KUKA KRL program: MyProgram_155().src

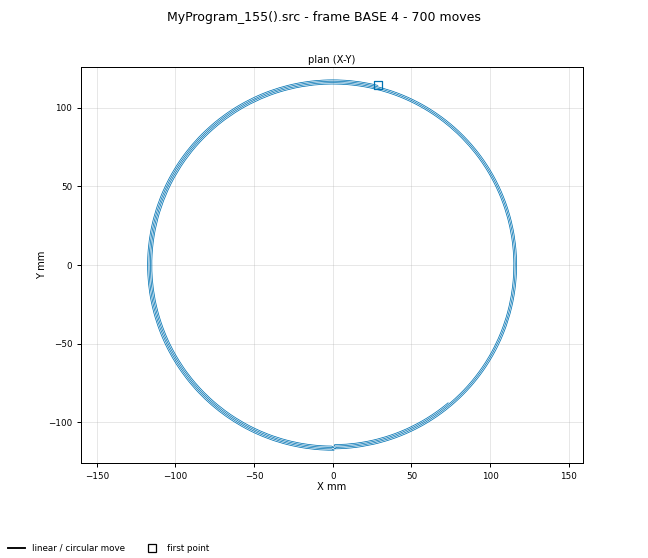
[picture p0: tool path of MyProgram_155().src in frame BASE 4, 700 of 700 moves have a stored position in this frame; points joined in program order, loops and branches not executed]
&ACCESS RVP
&REL 1
&PARAM TEMPLATE = C:\KRC\Roboter\Template\vorgabe
&PARAM EDITMASK = *
DEF MyProgram_155()
; ---- Setting reference (Base) ----
$BASE = BASE_DATA[4]

; --------------------------
; ---- Setting tool (TCP) ----
$TOOL = TOOL_DATA[3]
; --------------------------

$VEL.CP = VEL_APROX_PRINT
Startdeposition()
$VEL.CP = VEL_PRINT
LIN {X 28.6075,Y 114.2074,Z 120,A 72.0613,B 24.9358,C -1.85,E1 25.0377,E2 373.8713} C_DIS
LIN {X 25.7961,Y 114.8751,Z 120,A 73.4659,B 24.9358,C -1.8507,E1 25.0339,E2 372.4669} C_DIS
LIN {X 22.9691,Y 115.4736,Z 120,A 74.8709,B 24.9358,C -1.8512,E1 25.03,E2 371.0624} C_DIS
LIN {X 19.9429,Y 116.0335,Z 120,A 76.3004,B 24.9359,C -1.8487,E1 25.0261,E2 369.6403} C_DIS
LIN {X 17.2754,Y 116.4615,Z 120,A 77.5817,B 24.936,C -1.8476,E1 25.0226,E2 368.3629} C_DIS
LIN {X 14.0119,Y 116.8973,Z 120,A 79.1444,B 24.9361,C -1.8462,E1 25.0183,E2 366.8047} C_DIS
LIN {X 11.5401,Y 117.1689,Z 120,A 80.3543,B 24.9361,C -1.8463,E1 25.0149,E2 365.5954} C_DIS
LIN {X 8.2592,Y 117.444,Z 120,A 81.7792,B 24.9366,C -1.8385,E1 25.011,E2 364.1898} C_DIS
LIN {X 5.3745,Y 117.6113,Z 120,A 83.363,B 24.9361,C -1.8464,E1 25.0065,E2 362.5878} C_DIS
LIN {X 2.8894,Y 117.7004,Z 120,A 84.5732,B 24.9361,C -1.8462,E1 25.0032,E2 361.3782} C_DIS
LIN {X -0.4029,Y 117.7334,Z 120,A 85.999,B 24.9367,C -1.8381,E1 24.9992,E2 359.9717} C_DIS
LIN {X -3.2921,Y 117.688,Z 120,A 87.6216,B 24.936,C -1.8474,E1 24.9946,E2 358.3271} C_DIS
LIN {X -6.1794,Y 117.5718,Z 120,A 88.9298,B 24.9364,C -1.8425,E1 24.991,E2 357.03} C_DIS
LIN {X -9.0628,Y 117.3847,Z 120,A 90.3978,B 24.9362,C -1.8447,E1 24.9869,E2 355.5564} C_DIS
LIN {X -11.5401,Y 117.1689,Z 120,A 91.6095,B 24.9362,C -1.8441,E1 24.9835,E2 354.3454} C_DIS
LIN {X -14.4121,Y 116.8504,Z 120,A 93.1564,B 24.9359,C -1.8495,E1 24.9792,E2 352.7847} C_DIS
LIN {X -17.2754,Y 116.4615,Z 120,A 94.5644,B 24.9359,C -1.8486,E1 24.9753,E2 351.3776} C_DIS
LIN {X -20.1283,Y 116.0025,Z 120,A 95.973,B 24.936,C -1.8477,E1 24.9715,E2 349.9698} C_DIS
LIN {X -22.9691,Y 115.4736,Z 120,A 97.3817,B 24.936,C -1.8467,E1 24.9676,E2 348.5621} C_DIS
LIN {X -25.7961,Y 114.8751,Z 120,A 98.7906,B 24.9362,C -1.8455,E1 24.9638,E2 347.1541} C_DIS
LIN {X -28.6075,Y 114.2074,Z 120,A 100.1998,B 24.9362,C -1.8443,E1 24.9599,E2 345.7459} C_DIS
LIN {X -31.7893,Y 113.3611,Z 120,A 101.667,B 24.9368,C -1.8367,E1 24.956,E2 344.2943} C_DIS
LIN {X -34.1769,Y 112.6662,Z 120,A 103.0191,B 24.9364,C -1.8415,E1 24.9524,E2 342.9286} C_DIS
LIN {X -37.0459,Y 111.7549,Z 120,A 104.2953,B 24.9371,C -1.8316,E1 24.949,E2 341.6737} C_DIS
LIN {X -39.664,Y 110.8535,Z 120,A 105.7247,B 24.937,C -1.8334,E1 24.9453,E2 340.2371} C_DIS
LIN {X -42.3725,Y 109.8467,Z 120,A 107.2493,B 24.9368,C -1.8367,E1 24.9413,E2 338.7016} C_DIS
LIN {X -45.0555,Y 108.7737,Z 120,A 108.5208,B 24.9373,C -1.8288,E1 24.938,E2 337.4459} C_DIS
LIN {X -47.7114,Y 107.6352,Z 120,A 109.9314,B 24.9374,C -1.8269,E1 24.9344,E2 336.0364} C_DIS
LIN {X -50.68,Y 106.2678,Z 120,A 111.5717,B 24.9374,C -1.8266,E1 24.9302,E2 334.3928} C_DIS
LIN {X -53.2942,Y 104.9811,Z 120,A 112.9504,B 24.9377,C -1.8226,E1 24.9268,E2 333.0199} C_DIS
LIN {X -55.5003,Y 103.8337,Z 120,A 114.1649,B 24.9379,C -1.8207,E1 24.9238,E2 331.8065} C_DIS
LIN {X -58.0318,Y 102.4404,Z 120,A 115.5766,B 24.938,C -1.8185,E1 24.9204,E2 330.396} C_DIS
LIN {X -60.5283,Y 100.9854,Z 120,A 116.9884,B 24.9382,C -1.8162,E1 24.917,E2 328.9855} C_DIS
LIN {X -62.9884,Y 99.4695,Z 120,A 118.4003,B 24.9383,C -1.8138,E1 24.9137,E2 327.5749} C_DIS
LIN {X -65.4105,Y 97.8938,Z 120,A 119.9516,B 24.9381,C -1.8172,E1 24.91,E2 326.0103} C_DIS
LIN {X -68.1213,Y 96.025,Z 120,A 121.4219,B 24.9387,C -1.8083,E1 24.9067,E2 324.5561} C_DIS
LIN {X -70.4573,Y 94.3243,Z 120,A 122.8343,B 24.9389,C -1.8057,E1 24.9035,E2 323.145} C_DIS
LIN {X -72.4348,Y 92.8166,Z 120,A 124.0501,B 24.939,C -1.8033,E1 24.9008,E2 321.9305} C_DIS
LIN {X -74.6908,Y 91.011,Z 120,A 125.4632,B 24.9392,C -1.8005,E1 24.8978,E2 320.5187} C_DIS
LIN {X -76.9018,Y 89.1506,Z 120,A 126.8762,B 24.9394,C -1.7976,E1 24.8948,E2 319.1072} C_DIS
LIN {X -79.3634,Y 86.9641,Z 120,A 128.3082,B 24.9402,C -1.7867,E1 24.8918,E2 317.6952} C_DIS
LIN {X -81.1836,Y 85.2698,Z 120,A 129.7028,B 24.9398,C -1.7916,E1 24.889,E2 316.2833} C_DIS
LIN {X -83.2518,Y 83.2518,Z 120,A 131.2559,B 24.9397,C -1.7944,E1 24.8859,E2 314.7171} C_DIS
LIN {X -85.2976,Y 81.1541,Z 120,A 132.6747,B 24.9399,C -1.7905,E1 24.8831,E2 313.3013} C_DIS
LIN {X -87.5053,Y 78.7663,Z 120,A 134.1381,B 24.9405,C -1.7815,E1 24.8804,E2 311.8529} C_DIS
LIN {X -89.1506,Y 76.9018,Z 120,A 135.4975,B 24.9403,C -1.7846,E1 24.8779,E2 310.4799} C_DIS
LIN {X -91.2647,Y 74.3778,Z 120,A 136.9698,B 24.941,C -1.7749,E1 24.8753,E2 309.0239} C_DIS
LIN {X -92.8166,Y 72.4348,Z 120,A 138.1869,B 24.9412,C -1.772,E1 24.8732,E2 307.8081} C_DIS
LIN {X -94.5663,Y 70.1351,Z 120,A 139.7409,B 24.941,C -1.7743,E1 24.8706,E2 306.2411} C_DIS
LIN {X -96.259,Y 67.7932,Z 120,A 141.0161,B 24.9416,C -1.7649,E1 24.8685,E2 304.982} C_DIS
LIN {X -97.8938,Y 65.4105,Z 120,A 142.5702,B 24.9415,C -1.7672,E1 24.8661,E2 303.4147} C_DIS
LIN {X -99.4695,Y 62.9884,Z 120,A 143.9852,B 24.9417,C -1.7635,E1 24.864,E2 302.0013} C_DIS
LIN {X -101.1904,Y 60.1814,Z 120,A 145.2797,B 24.9429,C -1.7461,E1 24.8621,E2 300.7417} C_DIS
LIN {X -102.4404,Y 58.0318,Z 120,A 146.8155,B 24.9422,C -1.7561,E1 24.86,E2 299.1741} C_DIS
LIN {X -104.1352,Y 54.9278,Z 120,A 148.336,B 24.9431,C -1.7427,E1 24.858,E2 297.6775} C_DIS
LIN {X -105.8265,Y 51.5985,Z 120,A 150.2163,B 24.9433,C -1.7398,E1 24.8556,E2 295.7939} C_DIS
LIN {X -107.0416,Y 49.0287,Z 120,A 151.6575,B 24.9433,C -1.738,E1 24.8539,E2 294.3491} C_DIS
LIN {X -108.2126,Y 46.387,Z 120,A 153.1846,B 24.9433,C -1.7387,E1 24.8522,E2 292.8119} C_DIS
LIN {X -109.4657,Y 43.3423,Z 120,A 154.4796,B 24.9445,C -1.721,E1 24.8509,E2 291.5518} C_DIS
LIN {X -110.5368,Y 40.5322,Z 120,A 155.9008,B 24.9449,C -1.7147,E1 24.8495,E2 290.1376} C_DIS
LIN {X -111.3319,Y 38.3007,Z 120,A 157.3984,B 24.9442,C -1.7254,E1 24.8481,E2 288.6062} C_DIS
LIN {X -112.2383,Y 35.5569,Z 120,A 158.7082,B 24.9448,C -1.7169,E1 24.847,E2 287.309} C_DIS
LIN {X -113.2232,Y 32.2759,Z 120,A 160.3455,B 24.9452,C -1.7104,E1 24.8457,E2 285.6778} C_DIS
LIN {X -113.9481,Y 29.6166,Z 120,A 161.559,B 24.9458,C -1.7008,E1 24.8448,E2 284.48} C_DIS
LIN {X -114.5499,Y 27.2038,Z 120,A 163.0954,B 24.9452,C -1.7104,E1 24.8438,E2 282.9118} C_DIS
LIN {X -115.264,Y 23.9897,Z 120,A 164.3908,B 24.9463,C -1.6926,E1 24.8431,E2 281.6513} C_DIS
LIN {X -115.8181,Y 21.1538,Z 120,A 165.807,B 24.9466,C -1.6884,E1 24.8423,E2 280.2367} C_DIS
LIN {X -116.3023,Y 18.3051,Z 120,A 167.2233,B 24.9468,C -1.6843,E1 24.8417,E2 278.8218} C_DIS
LIN {X -116.6647,Y 15.845,Z 120,A 168.7598,B 24.9462,C -1.6938,E1 24.8411,E2 277.2534} C_DIS
LIN {X -117.0604,Y 12.5763,Z 120,A 170.0553,B 24.9474,C -1.6759,E1 24.8407,E2 275.9928} C_DIS
LIN {X -117.3017,Y 10.1014,Z 120,A 171.5922,B 24.9468,C -1.6855,E1 24.8403,E2 274.4239} C_DIS
LIN {X -117.5143,Y 7.2196,Z 120,A 173.0082,B 24.947,C -1.6813,E1 24.84,E2 273.0094} C_DIS
LIN {X -117.656,Y 4.3335,Z 120,A 174.4245,B 24.9473,C -1.6771,E1 24.8399,E2 271.5945} C_DIS
LIN {X -117.7313,Y 0.8208,Z 120,A 176.0503,B 24.9479,C -1.6681,E1 24.8398,E2 269.9803} C_DIS
LIN {X -117.7004,Y -2.8894,Z 120,A 177.825,B 24.9483,C -1.6609,E1 24.8398,E2 268.2121} C_DIS
LIN {X -117.5718,Y -6.1794,Z 120,A 179.2603,B 24.9491,C -1.6488,E1 24.84,E2 266.797} C_DIS
LIN {X -117.3847,Y -9.0628,Z 120,A -179.1455,B 24.9489,C -1.6521,E1 24.8403,E2 265.1855} C_DIS
LIN {X -117.1689,Y -11.5401,Z 120,A -177.9267,B 24.9491,C -1.6485,E1 24.8407,E2 263.9679} C_DIS
LIN {X -116.7986,Y -14.8117,Z 120,A -176.3132,B 24.9494,C -1.6439,E1 24.8412,E2 262.3558} C_DIS
LIN {X -116.4615,Y -17.2754,Z 120,A -174.9554,B 24.9492,C -1.6461,E1 24.8418,E2 260.9845} C_DIS
LIN {X -116.0025,Y -20.1283,Z 120,A -173.5394,B 24.9495,C -1.6421,E1 24.8424,E2 259.5697} C_DIS
LIN {X -115.4736,Y -22.9691,Z 120,A -172.1236,B 24.9497,C -1.638,E1 24.8432,E2 258.1553} C_DIS
LIN {X -114.7514,Y -26.3313,Z 120,A -170.5534,B 24.9503,C -1.6285,E1 24.8441,E2 256.5985} C_DIS
LIN {X -113.7427,Y -30.3958,Z 120,A -168.5264,B 24.9507,C -1.6217,E1 24.8455,E2 254.5758} C_DIS
LIN {X -112.9625,Y -33.178,Z 120,A -167.2894,B 24.9514,C -1.6104,E1 24.8464,E2 253.3588} C_DIS
LIN {X -112.1142,Y -35.9403,Z 120,A -165.8738,B 24.9516,C -1.6065,E1 24.8476,E2 251.9444} C_DIS
LIN {X -111.3319,Y -38.3007,Z 120,A -164.4772,B 24.9514,C -1.6106,E1 24.8489,E2 250.53} C_DIS
LIN {X -110.3584,Y -41.0214,Z 120,A -163.062,B 24.9516,C -1.6067,E1 24.8502,E2 249.1159} C_DIS
LIN {X -109.3184,Y -43.7173,Z 120,A -161.5073,B 24.9516,C -1.6088,E1 24.8518,E2 247.5475} C_DIS
LIN {X -108.2126,Y -46.387,Z 120,A -160.2317,B 24.9521,C -1.5993,E1 24.8532,E2 246.2877} C_DIS
LIN {X -107.0416,Y -49.0287,Z 120,A -158.8168,B 24.9523,C -1.5956,E1 24.8548,E2 244.8738} C_DIS
LIN {X -105.8062,Y -51.6408,Z 120,A -157.2625,B 24.9522,C -1.5978,E1 24.8567,E2 243.3057} C_DIS
LIN {X -104.3192,Y -54.5784,Z 120,A -155.9681,B 24.9532,C -1.5804,E1 24.8584,E2 242.0459} C_DIS
LIN {X -102.9484,Y -57.1221,Z 120,A -154.5537,B 24.9534,C -1.5769,E1 24.8602,E2 240.6325} C_DIS
LIN {X -101.7206,Y -59.2845,Z 120,A -152.9791,B 24.9527,C -1.5889,E1 24.8625,E2 239.0209} C_DIS
LIN {X -99.4695,Y -62.9884,Z 120,A -150.8974,B 24.9531,C -1.5822,E1 24.8655,E2 236.9446} C_DIS
LIN {X -97.6678,Y -65.7442,Z 120,A -149.4255,B 24.9537,C -1.5725,E1 24.8678,E2 235.4884} C_DIS
LIN {X -96.025,Y -68.1213,Z 120,A -148.0114,B 24.9539,C -1.5693,E1 24.8701,E2 234.075} C_DIS
LIN {X -94.3243,Y -70.4573,Z 120,A -146.5978,B 24.954,C -1.5661,E1 24.8724,E2 232.6622} C_DIS
LIN {X -92.8166,Y -72.4348,Z 120,A -145.3812,B 24.9542,C -1.5634,E1 24.8745,E2 231.4463} C_DIS
LIN {X -91.011,Y -74.6908,Z 120,A -143.8283,B 24.954,C -1.5663,E1 24.8772,E2 229.8793} C_DIS
LIN {X -88.8855,Y -77.2053,Z 120,A -142.5354,B 24.955,C -1.5494,E1 24.8795,E2 228.6207} C_DIS
LIN {X -87.2365,Y -79.0665,Z 120,A -141.0019,B 24.9544,C -1.5604,E1 24.8824,E2 227.0541} C_DIS
LIN {X -85.2698,Y -81.1836,Z 120,A -139.7283,B 24.9549,C -1.5516,E1 24.8849,E2 225.7959} C_DIS
LIN {X -82.9651,Y -83.535,Z 120,A -138.1185,B 24.9551,C -1.5485,E1 24.888,E2 224.1866} C_DIS
LIN {X -81.1836,Y -85.2698,Z 120,A -136.7639,B 24.9549,C -1.5522,E1 24.8908,E2 222.8176} C_DIS
LIN {X -78.7439,Y -87.5253,Z 120,A -135.4704,B 24.9559,C -1.535,E1 24.8934,E2 221.5598} C_DIS
LIN {X -76.8519,Y -89.1932,Z 120,A -133.931,B 24.9552,C -1.546,E1 24.8967,E2 219.9882} C_DIS
LIN {X -74.3778,Y -91.2647,Z 120,A -132.4694,B 24.9557,C -1.5384,E1 24.8998,E2 218.5392} C_DIS
LIN {X -72.2665,Y -92.9463,Z 120,A -131.2444,B 24.956,C -1.5321,E1 24.9025,E2 217.3247} C_DIS
LIN {X -70.1351,Y -94.5663,Z 120,A -129.7144,B 24.9556,C -1.5396,E1 24.9059,E2 215.7712} C_DIS
LIN {X -67.7933,Y -96.259,Z 120,A -128.4312,B 24.956,C -1.5319,E1 24.9088,E2 214.5021} C_DIS
LIN {X -65.3554,Y -97.9301,Z 120,A -126.873,B 24.9559,C -1.5348,E1 24.9125,E2 212.9318} C_DIS
LIN {X -62.9884,Y -99.4695,Z 120,A -125.6092,B 24.9563,C -1.5278,E1 24.9154,E2 211.6806} C_DIS
LIN {X -60.1814,Y -101.1904,Z 120,A -124.0018,B 24.9563,C -1.5257,E1 24.9193,E2 210.0732} C_DIS
LIN {X -57.994,Y -102.4615,Z 120,A -122.6437,B 24.9562,C -1.5295,E1 24.9226,E2 208.7021} C_DIS
LIN {X -55.5003,Y -103.8337,Z 120,A -121.3776,B 24.9566,C -1.5223,E1 24.9257,E2 207.4494} C_DIS
LIN {X -52.5743,Y -105.3435,Z 120,A -119.771,B 24.9566,C -1.5205,E1 24.9297,E2 205.8427} C_DIS
LIN {X -49.9732,Y -106.602,Z 120,A -118.361,B 24.9568,C -1.519,E1 24.9332,E2 204.4328} C_DIS
LIN {X -47.342,Y -107.7963,Z 120,A -117.1289,B 24.9573,C -1.5098,E1 24.9363,E2 203.2196} C_DIS
LIN {X -44.6823,Y -108.9256,Z 120,A -115.5421,B 24.9569,C -1.5163,E1 24.9404,E2 201.6138} C_DIS
LIN {X -41.8052,Y -110.0615,Z 120,A -114.0944,B 24.9572,C -1.5123,E1 24.9442,E2 200.1724} C_DIS
LIN {X -39.2838,Y -110.9869,Z 120,A -112.724,B 24.9571,C -1.5139,E1 24.9478,E2 198.7955} C_DIS
LIN {X -36.9316,Y -111.7935,Z 120,A -111.3729,B 24.9568,C -1.5192,E1 24.9514,E2 197.4294} C_DIS
LIN {X -33.9916,Y -112.7211,Z 120,A -109.9455,B 24.957,C -1.5148,E1 24.9552,E2 196.0098} C_DIS
LIN {X -31.4016,Y -113.471,Z 120,A -108.5562,B 24.9569,C -1.5174,E1 24.959,E2 194.6122} C_DIS
LIN {X -28.6075,Y -114.2074,Z 120,A -107.1484,B 24.9569,C -1.5166,E1 24.9628,E2 193.2041} C_DIS
LIN {X -25.7961,Y -114.8751,Z 120,A -105.7406,B 24.9569,C -1.516,E1 24.9666,E2 191.7961} C_DIS
LIN {X -22.9691,Y -115.4736,Z 120,A -104.3331,B 24.9569,C -1.5155,E1 24.9705,E2 190.3881} C_DIS
LIN {X -20.1283,Y -116.0025,Z 120,A -102.9258,B 24.9569,C -1.515,E1 24.9743,E2 188.9805} C_DIS
LIN {X -17.2754,Y -116.4615,Z 120,A -101.6573,B 24.9574,C -1.5084,E1 24.9778,E2 187.7265} C_DIS
LIN {X -14.0119,Y -116.8973,Z 120,A -100.0542,B 24.9574,C -1.5082,E1 24.9822,E2 186.1229} C_DIS
LIN {X -11.5401,Y -117.1689,Z 120,A -98.8438,B 24.9574,C -1.5081,E1 24.9856,E2 184.912} C_DIS
LIN {X -8.2592,Y -117.444,Z 120,A -97.3129,B 24.9576,C -1.5048,E1 24.9899,E2 183.3882} C_DIS
LIN {X -5.3745,Y -117.6113,Z 120,A -95.8351,B 24.9574,C -1.5082,E1 24.994,E2 181.9021} C_DIS
LIN {X -2.8894,Y -117.7004,Z 120,A -94.6255,B 24.9574,C -1.5082,E1 24.9974,E2 180.6921} C_DIS
LIN {X 0.8293,Y -117.7293,Z 120,A -93.0037,B 24.9578,C -1.5002,E1 25.0019,E2 179.0895} C_DIS
Enddeposition()
LIN {X 0.8293,Y -117.7293,Z 120,A -93.0037,B 24.9578,C -1.5002,E1 25.0019,E2 179.0895} C_DIS
Startdeposition()
$VEL.CP = VEL_PRINT
LIN {X -0.5833,Y -116.846,Z 120,A -94.2822,B 24.9585,C -1.4892,E1 24.9982,E2 180.394} C_DIS
LIN {X -3.7681,Y -116.7867,Z 120,A -95.7825,B 24.9583,C -1.4917,E1 24.994,E2 181.8886} C_DIS
LIN {X -6.6179,Y -116.6599,Z 120,A -97.1718,B 24.9583,C -1.492,E1 24.9902,E2 183.2775} C_DIS
LIN {X -9.8038,Y -116.4364,Z 120,A -98.8453,B 24.9586,C -1.4872,E1 24.9855,E2 184.963} C_DIS
LIN {X -13.6561,Y -116.0466,Z 120,A -100.6924,B 24.9584,C -1.4898,E1 24.9804,E2 186.8052} C_DIS
LIN {X -17.4959,Y -115.5306,Z 120,A -102.5961,B 24.9584,C -1.49,E1 24.9751,E2 188.7098} C_DIS
LIN {X -20.8591,Y -114.9706,Z 120,A -104.2133,B 24.9582,C -1.493,E1 24.9707,E2 190.3216} C_DIS
LIN {X -24.4922,Y -114.2524,Z 120,A -106.1589,B 24.9585,C -1.4881,E1 24.9653,E2 192.2812} C_DIS
LIN {X -27.6951,Y -113.5178,Z 120,A -107.672,B 24.9582,C -1.4932,E1 24.9612,E2 193.7841} C_DIS
LIN {X -30.8948,Y -112.6899,Z 120,A -109.1999,B 24.9579,C -1.4983,E1 24.9571,E2 195.3023} C_DIS
LIN {X -33.8766,Y -111.8301,Z 120,A -111.8951,B 24.9607,C -1.4487,E1 24.9496,E2 198.1197} C_DIS
LIN {X -40.072,Y -109.7613,Z 120,A -113.983,B 24.9579,C -1.4994,E1 24.9444,E2 200.0914} C_DIS
LIN {X -43.4727,Y -108.4612,Z 120,A -115.8418,B 24.9579,C -1.4979,E1 24.9395,E2 201.9578} C_DIS
LIN {X -47.2007,Y -106.8911,Z 120,A -117.7204,B 24.9576,C -1.5046,E1 24.9348,E2 203.8249} C_DIS
LIN {X -49.4784,Y -105.8548,Z 120,A -119.1132,B 24.9579,C -1.4989,E1 24.9312,E2 205.2347} C_DIS
LIN {X -53.1358,Y -104.0668,Z 120,A -120.8787,B 24.9572,C -1.5113,E1 24.9268,E2 206.9753} C_DIS
LIN {X -56.434,Y -102.3176,Z 120,A -122.7584,B 24.9572,C -1.5116,E1 24.9222,E2 208.8596} C_DIS
LIN {X -59.1122,Y -100.7929,Z 120,A -124.3925,B 24.9574,C -1.5085,E1 24.9182,E2 210.5059} C_DIS
LIN {X -61.827,Y -99.1501,Z 120,A -125.9835,B 24.9574,C -1.5094,E1 24.9144,E2 212.0998} C_DIS
LIN {X -65.022,Y -97.0865,Z 120,A -127.9181,B 24.9574,C -1.5094,E1 24.9099,E2 214.0408} C_DIS
LIN {X -68.4014,Y -94.7364,Z 120,A -130.2054,B 24.9578,C -1.5014,E1 24.9046,E2 216.3548} C_DIS
LIN {X -71.0173,Y -92.7901,Z 120,A -131.2356,B 24.9562,C -1.5284,E1 24.9025,E2 217.3248} C_DIS
LIN {X -73.512,Y -90.8256,Z 120,A -133.0468,B 24.9567,C -1.5205,E1 24.8985,E2 219.1614} C_DIS
LIN {X -76.9746,Y -87.9104,Z 120,A -135.1903,B 24.9563,C -1.528,E1 24.8939,E2 221.2953} C_DIS
LIN {X -79.5354,Y -85.6032,Z 120,A -136.9573,B 24.9563,C -1.5282,E1 24.8903,E2 223.0691} C_DIS
LIN {X -83.7073,Y -81.5277,Z 120,A -139.6988,B 24.9556,C -1.5392,E1 24.8849,E2 225.7958} C_DIS
LIN {X -86.2695,Y -78.8096,Z 120,A -141.6709,B 24.9557,C -1.5374,E1 24.8811,E2 227.7808} C_DIS
LIN {X -89.6384,Y -74.956,Z 120,A -144.2184,B 24.9555,C -1.5417,E1 24.8764,E2 230.3298} C_DIS
LIN {X -91.9256,Y -72.1328,Z 120,A -146.5553,B 24.9565,C -1.523,E1 24.8723,E2 232.7221} C_DIS
LIN {X -94.566,Y -68.6354,Z 120,A -148.019,B 24.9546,C -1.5567,E1 24.87,E2 234.1128} C_DIS
LIN {X -95.9693,Y -66.6574,Z 120,A -149.3147,B 24.9546,C -1.5553,E1 24.8679,E2 235.4182} C_DIS
LIN {X -98.1483,Y -63.406,Z 120,A -151.5108,B 24.9551,C -1.5488,E1 24.8645,E2 237.6406} C_DIS
LIN {X -100.0436,Y -60.3715,Z 120,A -153.0221,B 24.9542,C -1.5635,E1 24.8623,E2 239.1247} C_DIS
LIN {X -102.1243,Y -56.7802,Z 120,A -155.075,B 24.9539,C -1.5683,E1 24.8595,E2 241.1769} C_DIS
LIN {X -104.1156,Y -53.0403,Z 120,A -157.1484,B 24.9536,C -1.5743,E1 24.8568,E2 243.2472} C_DIS
LIN {X -105.5963,Y -50.0314,Z 120,A -158.9261,B 24.9536,C -1.5734,E1 24.8546,E2 245.0364} C_DIS
LIN {X -108.1129,Y -44.3283,Z 120,A -161.6818,B 24.9524,C -1.5946,E1 24.8516,E2 247.7568} C_DIS
LIN {X -108.9291,Y -42.2844,Z 120,A -162.8718,B 24.9524,C -1.5933,E1 24.8504,E2 248.9568} C_DIS
LIN {X -109.8159,Y -39.9223,Z 120,A -164.2194,B 24.9524,C -1.5924,E1 24.8491,E2 250.314} C_DIS
LIN {X -111.2193,Y -35.8272,Z 120,A -166.3646,B 24.9522,C -1.5979,E1 24.8472,E2 252.4583} C_DIS
LIN {X -112.4296,Y -31.8258,Z 120,A -168.4471,B 24.9519,C -1.6029,E1 24.8455,E2 254.541} C_DIS
LIN {X -113.5161,Y -27.702,Z 120,A -170.5072,B 24.9514,C -1.6106,E1 24.8441,E2 256.5947} C_DIS
LIN {X -114.2632,Y -24.4427,Z 120,A -172.1219,B 24.951,C -1.6167,E1 24.8431,E2 258.2043} C_DIS
LIN {X -114.9448,Y -21.0025,Z 120,A -173.8973,B 24.9508,C -1.6199,E1 24.8422,E2 259.9827} C_DIS
LIN {X -115.8291,Y -15.3974,Z 120,A -176.4915,B 24.9498,C -1.6364,E1 24.8411,E2 262.553} C_DIS
LIN {X -116.295,Y -11.3652,Z 120,A -178.8276,B 24.9503,C -1.6287,E1 24.8404,E2 264.9214} C_DIS
LIN {X -116.6596,Y -6.6243,Z 120,A 178.8642,B 24.9498,C -1.6372,E1 24.84,E2 267.2232} C_DIS
LIN {X -116.8144,Y -2.8659,Z 120,A 177.0384,B 24.9494,C -1.6439,E1 24.8398,E2 269.044} C_DIS
LIN {X -116.8438,Y 0.9933,Z 120,A 175.1495,B 24.949,C -1.6503,E1 24.8398,E2 270.9291} C_DIS
LIN {X -116.7276,Y 5.2971,Z 120,A 172.8004,B 24.9491,C -1.6476,E1 24.84,E2 273.2989} C_DIS
LIN {X -116.489,Y 9.1463,Z 120,A 171.1669,B 24.9481,C -1.6641,E1 24.8404,E2 274.9027} C_DIS
LIN {X -115.8711,Y 15.0729,Z 120,A 168.3215,B 24.9473,C -1.6767,E1 24.8413,E2 277.7351} C_DIS
LIN {X -115.1266,Y 19.9815,Z 120,A 165.8287,B 24.947,C -1.6822,E1 24.8423,E2 280.2296} C_DIS
LIN {X -114.6957,Y 22.3215,Z 120,A 164.015,B 24.9484,C -1.6599,E1 24.8433,E2 282.1071} C_DIS
LIN {X -113.8096,Y 26.4711,Z 120,A 161.8481,B 24.9482,C -1.6632,E1 24.8447,E2 284.2791} C_DIS
LIN {X -112.6767,Y 30.9437,Z 120,A 160.3303,B 24.9458,C -1.7004,E1 24.8457,E2 285.717} C_DIS
LIN {X -111.952,Y 33.4681,Z 120,A 158.9357,B 24.9458,C -1.7001,E1 24.8468,E2 287.1203} C_DIS
LIN {X -110.6888,Y 37.4339,Z 120,A 156.8632,B 24.9455,C -1.7053,E1 24.8486,E2 289.1923} C_DIS
LIN {X -109.648,Y 40.3826,Z 120,A 155.3478,B 24.9451,C -1.7108,E1 24.8501,E2 290.7031} C_DIS
LIN {X -108.6603,Y 42.9688,Z 120,A 153.8954,B 24.9451,C -1.7112,E1 24.8515,E2 292.1628} C_DIS
LIN {X -106.5918,Y 47.8697,Z 120,A 151.318,B 24.9445,C -1.7204,E1 24.8544,E2 294.7323} C_DIS
LIN {X -104.0815,Y 53.1071,Z 120,A 148.8034,B 24.9431,C -1.7426,E1 24.8574,E2 297.2078} C_DIS
LIN {X -102.348,Y 56.3794,Z 120,A 146.3255,B 24.9445,C -1.721,E1 24.8608,E2 299.7503} C_DIS
LIN {X -99.8932,Y 60.619,Z 120,A 144.2276,B 24.9432,C -1.7403,E1 24.8637,E2 301.8129} C_DIS
LIN {X -98.0409,Y 63.5734,Z 120,A 142.3789,B 24.9432,C -1.7395,E1 24.8665,E2 303.6729} C_DIS
LIN {X -95.9693,Y 66.6573,Z 120,A 140.6979,B 24.9426,C -1.7504,E1 24.8691,E2 305.3364} C_DIS
LIN {X -94.0429,Y 69.3499,Z 120,A 138.873,B 24.9428,C -1.7466,E1 24.8721,E2 307.1791} C_DIS
LIN {X -91.7233,Y 72.3888,Z 120,A 137.1219,B 24.9422,C -1.7567,E1 24.8751,E2 308.9144} C_DIS
LIN {X -89.8293,Y 74.7262,Z 120,A 135.7036,B 24.9417,C -1.763,E1 24.8776,E2 310.3244} C_DIS
LIN {X -87.5284,Y 77.4112,Z 120,A 133.9937,B 24.9414,C -1.7684,E1 24.8807,E2 312.0291} C_DIS
LIN {X -85.3016,Y 79.8562,Z 120,A 132.1845,B 24.9416,C -1.7648,E1 24.8842,E2 313.8548} C_DIS
LIN {X -82.6638,Y 82.586,Z 120,A 130.4757,B 24.9409,C -1.7756,E1 24.8875,E2 315.5452} C_DIS
LIN {X -80.9252,Y 84.288,Z 120,A 129.2342,B 24.9409,C -1.7765,E1 24.89,E2 316.7897} C_DIS
LIN {X -78.1093,Y 86.9039,Z 120,A 127.2894,B 24.9407,C -1.7785,E1 24.894,E2 318.7378} C_DIS
LIN {X -75.4686,Y 89.2074,Z 120,A 125.5023,B 24.9407,C -1.7795,E1 24.8978,E2 320.5293} C_DIS
LIN {X -72.6669,Y 91.5035,Z 120,A 123.7905,B 24.9402,C -1.7861,E1 24.9015,E2 322.2319} C_DIS
LIN {X -70.0802,Y 93.4991,Z 120,A 122.1557,B 24.9401,C -1.7881,E1 24.9051,E2 323.8678} C_DIS
LIN {X -67.4078,Y 95.4453,Z 120,A 120.6158,B 24.9396,C -1.7948,E1 24.9086,E2 325.3971} C_DIS
LIN {X -64.938,Y 97.1434,Z 120,A 119.1614,B 24.9394,C -1.7984,E1 24.912,E2 326.848} C_DIS
LIN {X -62.4604,Y 98.7544,Z 120,A 117.7195,B 24.9392,C -1.8015,E1 24.9153,E2 328.2871} C_DIS
LIN {X -59.4234,Y 100.609,Z 120,A 115.8698,B 24.9392,C -1.8003,E1 24.9198,E2 330.1451} C_DIS
LIN {X -56.786,Y 102.121,Z 120,A 114.3615,B 24.9392,C -1.8022,E1 24.9234,E2 331.6534} C_DIS
LIN {X -52.8753,Y 104.1999,Z 120,A 112.1336,B 24.939,C -1.8035,E1 24.929,E2 333.8843} C_DIS
LIN {X -45.1093,Y 107.7893,Z 120,A 107.9624,B 24.9385,C -1.8109,E1 24.9396,E2 338.0482} C_DIS
LIN {X -41.3286,Y 109.2943,Z 120,A 105.9734,B 24.9383,C -1.8139,E1 24.9447,E2 340.0344} C_DIS
LIN {X -38.0207,Y 110.4907,Z 120,A 104.1491,B 24.9385,C -1.8118,E1 24.9496,E2 341.8672} C_DIS
LIN {X -34.1404,Y 111.7496,Z 120,A 102.3429,B 24.9377,C -1.8224,E1 24.9543,E2 343.6513} C_DIS
LIN {X -31.8168,Y 112.4322,Z 120,A 101.0929,B 24.9378,C -1.821,E1 24.9577,E2 344.9066} C_DIS
LIN {X -28.5613,Y 113.3042,Z 120,A 99.1236,B 24.9386,C -1.8092,E1 24.9631,E2 346.9069} C_DIS
LIN {X -24.5198,Y 114.2464,Z 120,A 97.4082,B 24.9376,C -1.8247,E1 24.9677,E2 348.5877} C_DIS
LIN {X -20.8546,Y 114.9714,Z 120,A 95.5404,B 24.9376,C -1.8247,E1 24.9728,E2 350.4578} C_DIS
LIN {X -17.7549,Y 115.4906,Z 120,A 93.9865,B 24.9376,C -1.8252,E1 24.9771,E2 352.0118} C_DIS
LIN {X -13.8207,Y 116.0273,Z 120,A 91.9759,B 24.9376,C -1.8236,E1 24.9827,E2 354.0274} C_DIS
LIN {X -9.9632,Y 116.4237,Z 120,A 89.9577,B 24.9379,C -1.8195,E1 24.9883,E2 356.0565} C_DIS
LIN {X -6.0564,Y 116.691,Z 120,A 88.1401,B 24.9376,C -1.8247,E1 24.9933,E2 357.8624} C_DIS
LIN {X -1.865,Y 116.8328,Z 120,A 86.2333,B 24.9371,C -1.8318,E1 24.9986,E2 359.7526} C_DIS
LIN {X 0.9122,Y 116.844,Z 120,A 84.7627,B 24.9374,C -1.8273,E1 25.0028,E2 361.2337} C_DIS
LIN {X 4.2907,Y 116.7707,Z 120,A 83.2064,B 24.9371,C -1.8318,E1 25.0071,E2 362.779} C_DIS
LIN {X 7.6392,Y 116.5976,Z 120,A 81.5607,B 24.9371,C -1.8318,E1 25.0117,E2 364.4241} C_DIS
LIN {X 11.0317,Y 116.3258,Z 120,A 79.9381,B 24.937,C -1.8337,E1 25.0162,E2 366.0413} C_DIS
LIN {X 13.9759,Y 116.0092,Z 120,A 78.4496,B 24.9371,C -1.8318,E1 25.0203,E2 367.5332} C_DIS
LIN {X 17.163,Y 115.5821,Z 120,A 76.8742,B 24.9371,C -1.8314,E1 25.0246,E2 369.1081} C_DIS
LIN {X 20.0634,Y 115.1137,Z 120,A 75.4406,B 24.9371,C -1.8313,E1 25.0286,E2 370.5407} C_DIS
LIN {X 23.5374,Y 114.4522,Z 120,A 73.644,B 24.9374,C -1.8278,E1 25.0335,E2 372.3434} C_DIS
LIN {X 27.1678,Y 113.6464,Z 120,A 71.6794,B 24.9379,C -1.8205,E1 25.0389,E2 374.3224} C_DIS
LIN {X 31.2326,Y 112.5971,Z 120,A 68.7019,B 24.9407,C -1.7787,E1 25.0472,E2 377.3941} C_DIS
LIN {X 37.3634,Y 110.7126,Z 120,A 67.0087,B 24.9365,C -1.8405,E1 25.0513,E2 378.9378} C_DIS
LIN {X 41.4792,Y 109.2373,Z 120,A 64.5211,B 24.9377,C -1.823,E1 25.0579,E2 381.4616} C_DIS
LIN {X 44.7935,Y 107.9224,Z 120,A 62.8297,B 24.9377,C -1.8238,E1 25.0623,E2 383.1474} C_DIS
LIN {X 47.7574,Y 106.6424,Z 120,A 61.1868,B 24.938,C -1.8193,E1 25.0665,E2 384.7969} C_DIS
LIN {X 50.6964,Y 105.2767,Z 120,A 59.5747,B 24.9382,C -1.8164,E1 25.0706,E2 386.4118} C_DIS
LIN {X 54.3776,Y 103.4233,Z 120,A 57.5526,B 24.9383,C -1.8137,E1 25.0756,E2 388.4348} C_DIS
LIN {X 57.1544,Y 101.9153,Z 120,A 55.9552,B 24.9386,C -1.8093,E1 25.0795,E2 390.0378} C_DIS
LIN {X 59.9972,Y 100.2698,Z 120,A 54.47,B 24.9384,C -1.8126,E1 25.0831,E2 391.5107} C_DIS
LIN {X 62.2868,Y 98.8628,Z 120,A 52.9851,B 24.9391,C -1.803,E1 25.0866,E2 393.0136} C_DIS
LIN {X 65.5013,Y 96.762,Z 120,A 51.2606,B 24.9388,C -1.8071,E1 25.0906,E2 394.7225} C_DIS
LIN {X 68.9644,Y 94.3251,Z 120,A 49.171,B 24.9391,C -1.8029,E1 25.0954,E2 396.8147} C_DIS
LIN {X 71.7757,Y 92.2056,Z 120,A 47.3327,B 24.9396,C -1.7946,E1 25.0995,E2 398.6659} C_DIS
LIN {X 74.6746,Y 89.8722,Z 120,A 45.6175,B 24.9396,C -1.7962,E1 25.1031,E2 400.3709} C_DIS
LIN {X 77.4613,Y 87.484,Z 120,A 43.9093,B 24.9395,C -1.7968,E1 25.1067,E2 402.0709} C_DIS
LIN {X 79.9413,Y 85.2215,Z 120,A 42.0637,B 24.9403,C -1.7842,E1 25.1106,E2 403.9387} C_DIS
LIN {X 83.0621,Y 82.1827,Z 120,A 39.9987,B 24.9404,C -1.7829,E1 25.1146,E2 405.9981} C_DIS
LIN {X 86.1353,Y 78.9558,Z 120,A 37.9564,B 24.9404,C -1.7846,E1 25.1185,E2 408.0274} C_DIS
LIN {X 88.394,Y 76.4209,Z 120,A 36.1064,B 24.9411,C -1.7722,E1 25.122,E2 409.8986} C_DIS
LIN {X 90.883,Y 73.4412,Z 120,A 34.3936,B 24.9408,C -1.7765,E1 25.125,E2 411.5932} C_DIS
LIN {X 92.7846,Y 71.0244,Z 120,A 32.9119,B 24.941,C -1.7741,E1 25.1275,E2 413.0737} C_DIS
LIN {X 94.5189,Y 68.6997,Z 120,A 31.4706,B 24.9413,C -1.7696,E1 25.1299,E2 414.5186} C_DIS
LIN {X 96.2888,Y 66.1978,Z 120,A 29.9752,B 24.9415,C -1.7661,E1 25.1323,E2 416.015} C_DIS
LIN {X 98.2987,Y 63.1718,Z 120,A 28.1702,B 24.9419,C -1.7604,E1 25.1351,E2 417.8245} C_DIS
LIN {X 100.0635,Y 60.3388,Z 120,A 26.4162,B 24.9426,C -1.7505,E1 25.1377,E2 419.5929} C_DIS
LIN {X 102.1404,Y 56.7513,Z 120,A 24.5377,B 24.9425,C -1.7522,E1 25.1402,E2 421.4576} C_DIS
LIN {X 103.7357,Y 53.7836,Z 120,A 22.7222,B 24.9433,C -1.7399,E1 25.1426,E2 423.2926} C_DIS
LIN {X 105.5627,Y 50.1012,Z 120,A 20.8355,B 24.9433,C -1.7402,E1 25.1449,E2 425.1684} C_DIS
LIN {X 107.0832,Y 46.76,Z 120,A 19.0772,B 24.9435,C -1.737,E1 25.1469,E2 426.9246} C_DIS
LIN {X 108.3952,Y 43.6347,Z 120,A 17.3018,B 24.9441,C -1.7268,E1 25.1488,E2 428.7145} C_DIS
LIN {X 109.831,Y 39.8808,Z 120,A 15.4704,B 24.9441,C -1.7275,E1 25.1506,E2 430.5339} C_DIS
LIN {X 111.0216,Y 36.4382,Z 120,A 13.6818,B 24.9444,C -1.7219,E1 25.1522,E2 432.3255} C_DIS
LIN {X 112.6061,Y 31.2032,Z 120,A 11.0755,B 24.9447,C -1.7173,E1 25.1543,E2 434.9279} C_DIS
LIN {X 113.4315,Y 28.0487,Z 120,A 9.3537,B 24.9454,C -1.7065,E1 25.1554,E2 436.6651} C_DIS
LIN {X 114.629,Y 22.668,Z 120,A 6.8322,B 24.9454,C -1.7065,E1 25.1569,E2 439.1718} C_DIS
LIN {X 115.2494,Y 19.2584,Z 120,A 5.1751,B 24.9456,C -1.7032,E1 25.1577,E2 440.8271} C_DIS
LIN {X 115.736,Y 16.0814,Z 120,A 3.5366,B 24.9461,C -1.6952,E1 25.1584,E2 442.4749} C_DIS
LIN {X 116.0749,Y 13.4148,Z 120,A 2.1386,B 24.9467,C -1.6872,E1 25.1589,E2 443.8835} C_DIS
LIN {X 116.4326,Y 9.8516,Z 120,A 0.333,B 24.9472,C -1.6791,E1 25.1593,E2 445.6974} C_DIS
LIN {X 116.706,Y 5.7829,Z 120,A -1.5154,B 24.9472,C -1.6798,E1 25.1596,E2 447.5332} C_DIS
LIN {X 116.8262,Y 2.2252,Z 120,A -3.2494,B 24.9474,C -1.6747,E1 25.1598,E2 449.2688} C_DIS
LIN {X 116.8444,Y -0.9066,Z 120,A -4.8734,B 24.948,C -1.6655,E1 25.1598,E2 450.905} C_DIS
LIN {X 116.7547,Y -4.6655,Z 120,A -6.6816,B 24.9483,C -1.6612,E1 25.1596,E2 452.7126} C_DIS
LIN {X 116.5641,Y -8.1348,Z 120,A -8.2955,B 24.9483,C -1.6599,E1 25.1593,E2 454.3199} C_DIS
LIN {X 116.2375,Y -11.9247,Z 120,A -10.267,B 24.9491,C -1.6487,E1 25.1588,E2 456.306} C_DIS
LIN {X 115.8155,Y -15.502,Z 120,A -11.9375,B 24.9491,C -1.6475,E1 25.1582,E2 457.9695} C_DIS
LIN {X 115.2143,Y -19.4681,Z 120,A -13.8931,B 24.9495,C -1.6417,E1 25.1574,E2 459.9274} C_DIS
LIN {X 114.5137,Y -23.2378,Z 120,A -15.8606,B 24.9501,C -1.6314,E1 25.1563,E2 461.9077} C_DIS
LIN {X 113.7181,Y -26.867,Z 120,A -17.5141,B 24.95,C -1.6335,E1 25.1553,E2 463.5465} C_DIS
LIN {X 112.6239,Y -31.1383,Z 120,A -19.7934,B 24.9508,C -1.621,E1 25.1537,E2 465.8423} C_DIS
LIN {X 110.3423,Y -38.444,Z 120,A -23.1865,B 24.9504,C -1.6262,E1 25.1509,E2 469.2038} C_DIS
LIN {X 109.2096,Y -41.5523,Z 120,A -24.9615,B 24.9512,C -1.6139,E1 25.1491,E2 470.998} C_DIS
LIN {X 108.13,Y -44.2861,Z 120,A -26.4488,B 24.9516,C -1.6072,E1 25.1475,E2 472.4929} C_DIS
LIN {X 106.866,Y -47.2582,Z 120,A -27.993,B 24.9518,C -1.6042,E1 25.1458,E2 474.0357} C_DIS
LIN {X 105.1664,Y -50.926,Z 120,A -29.9821,B 24.9522,C -1.5978,E1 25.1435,E2 476.0291} C_DIS
LIN {X 103.6285,Y -53.9881,Z 120,A -31.7762,B 24.9528,C -1.5873,E1 25.1412,E2 477.8384} C_DIS
LIN {X 101.7027,Y -57.5351,Z 120,A -33.6106,B 24.9528,C -1.5883,E1 25.1387,E2 479.6608} C_DIS
LIN {X 99.513,Y -61.2445,Z 120,A -35.9382,B 24.9537,C -1.572,E1 25.1353,E2 482.0151} C_DIS
LIN {X 97.287,Y -64.7208,Z 120,A -37.7017,B 24.9533,C -1.5785,E1 25.1327,E2 483.7543} C_DIS
LIN {X 95.6658,Y -67.094,Z 120,A -39.2548,B 24.9539,C -1.5678,E1 25.1302,E2 485.3252} C_DIS
LIN {X 93.5067,Y -70.0701,Z 120,A -40.9629,B 24.9539,C -1.5673,E1 25.1273,E2 487.0262} C_DIS
LIN {X 91.4362,Y -72.7521,Z 120,A -42.5477,B 24.954,C -1.5664,E1 25.1246,E2 488.6057} C_DIS
LIN {X 89.6985,Y -74.8836,Z 120,A -43.9334,B 24.9543,C -1.561,E1 25.1222,E2 489.9976} C_DIS
LIN {X 87.6493,Y -77.2736,Z 120,A -45.6547,B 24.9551,C -1.5486,E1 25.119,E2 491.7404} C_DIS
LIN {X 85.02,Y -80.1556,Z 120,A -47.4183,B 24.9549,C -1.5508,E1 25.1156,E2 493.4911} C_DIS
LIN {X 82.8816,Y -82.3655,Z 120,A -48.8658,B 24.9549,C -1.5499,E1 25.1128,E2 494.9346} C_DIS
LIN {X 80.7786,Y -84.4293,Z 120,A -50.3175,B 24.9552,C -1.546,E1 25.1099,E2 496.3893} C_DIS
LIN {X 77.9121,Y -87.0805,Z 120,A -52.2096,B 24.9554,C -1.5426,E1 25.106,E2 498.282} C_DIS
LIN {X 75.251,Y -89.3928,Z 120,A -53.9799,B 24.9558,C -1.5366,E1 25.1022,E2 500.0595} C_DIS
LIN {X 71.7046,Y -92.2604,Z 120,A -56.0297,B 24.9555,C -1.5404,E1 25.0978,E2 502.0926} C_DIS
LIN {X 69.0016,Y -94.2979,Z 120,A -57.7276,B 24.9559,C -1.5351,E1 25.094,E2 503.797} C_DIS
LIN {X 66.1962,Y -96.2899,Z 120,A -59.6718,B 24.9567,C -1.5196,E1 25.0895,E2 505.771} C_DIS
LIN {X 63.0417,Y -98.3822,Z 120,A -61.3506,B 24.9565,C -1.5242,E1 25.0856,E2 507.4334} C_DIS
LIN {X 60.5918,Y -99.9097,Z 120,A -62.8103,B 24.9567,C -1.5195,E1 25.0821,E2 508.8997} C_DIS
LIN {X 56.9383,Y -102.036,Z 120,A -64.8888,B 24.957,C -1.5154,E1 25.077,E2 510.9815} C_DIS
LIN {X 52.5672,Y -104.3573,Z 120,A -67.1898,B 24.9569,C -1.5171,E1 25.0714,E2 513.2723} C_DIS
LIN {X 49.9029,Y -105.6572,Z 120,A -68.8175,B 24.9575,C -1.5067,E1 25.0672,E2 514.9202} C_DIS
LIN {X 46.5474,Y -107.1759,Z 120,A -70.4321,B 24.9571,C -1.5128,E1 25.0631,E2 516.5166} C_DIS
LIN {X 43.3491,Y -108.5109,Z 120,A -72.4244,B 24.958,C -1.4968,E1 25.0579,E2 518.542} C_DIS
LIN {X 39.8099,Y -109.8569,Z 120,A -74.0447,B 24.9576,C -1.5052,E1 25.0537,E2 520.1391} C_DIS
LIN {X 36.9308,Y -110.8585,Z 120,A -75.4859,B 24.9576,C -1.5057,E1 25.0499,E2 521.5762} C_DIS
LIN {X 33.5651,Y -111.9232,Z 120,A -78.0528,B 24.9598,C -1.4658,E1 25.0428,E2 524.233} C_DIS
LIN {X 28.5023,Y -113.3194,Z 120,A -79.7676,B 24.9577,C -1.502,E1 25.0384,E2 525.8596} C_DIS
LIN {X 25.9397,Y -113.9323,Z 120,A -81.2094,B 24.9582,C -1.4939,E1 25.0345,E2 527.3185} C_DIS
LIN {X 18.55,Y -115.3669,Z 120,A -84.9165,B 24.9584,C -1.4901,E1 25.0243,E2 531.0302} C_DIS
LIN {X 15.0044,Y -115.88,Z 120,A -86.5189,B 24.9581,C -1.4959,E1 25.0199,E2 532.6175} C_DIS
LIN {X 11.8631,Y -116.244,Z 120,A -88.0621,B 24.9581,C -1.4953,E1 25.0156,E2 534.1611} C_DIS
LIN {X 8.4545,Y -116.5425,Z 120,A -89.8195,B 24.9584,C -1.4909,E1 25.0107,E2 535.9281} C_DIS
LIN {X 4.829,Y -116.7477,Z 120,A -91.5864,B 24.9584,C -1.4909,E1 25.0057,E2 537.6945} C_DIS
LIN {X 0.8282,Y -116.8442,Z 120,A -93.4643,B 24.9582,C -1.4941,E1 25.0005,E2 539.5645} C_DIS
Enddeposition()
LIN {X 0.8282,Y -116.8442,Z 120,A -93.4643,B 24.9582,C -1.4941,E1 25.0005,E2 539.5645} C_DIS
Startdeposition()
$VEL.CP = VEL_PRINT
LIN {X 2.2203,Y -115.9399,Z 120,A -92.1188,B 24.9556,C -1.5392,E1 25.0046,E2 538.1122} C_DIS
LIN {X 6.9272,Y -115.7552,Z 120,A -89.8563,B 24.9557,C -1.5372,E1 25.0109,E2 535.8552} C_DIS
LIN {X 11.3845,Y -115.4028,Z 120,A -87.6729,B 24.9557,C -1.5372,E1 25.017,E2 533.6732} C_DIS
LIN {X 14.1565,Y -115.0957,Z 120,A -86.0615,B 24.9551,C -1.5485,E1 25.0215,E2 532.0359} C_DIS
LIN {X 19.8501,Y -114.2504,Z 120,A -82.6291,B 24.9534,C -1.5777,E1 25.0311,E2 528.538} C_DIS
LIN {X 24.7764,Y -113.2833,Z 120,A -80.9011,B 24.9553,C -1.5454,E1 25.0356,E2 526.8887} C_DIS
LIN {X 27.3361,Y -112.6931,Z 120,A -79.5399,B 24.955,C -1.5495,E1 25.0393,E2 525.5197} C_DIS
LIN {X 33.4498,Y -111.033,Z 120,A -76.6062,B 24.9553,C -1.5439,E1 25.0472,E2 522.604} C_DIS
LIN {X 36.2055,Y -110.1654,Z 120,A -75.0438,B 24.9549,C -1.5518,E1 25.0514,E2 521.0258} C_DIS
LIN {X 39.6716,Y -108.964,Z 120,A -73.2706,B 24.9549,C -1.5524,E1 25.056,E2 519.2548} C_DIS
LIN {X 44.5957,Y -107.0441,Z 120,A -70.8045,B 24.955,C -1.5494,E1 25.0624,E2 516.8014} C_DIS
LIN {X 47.4117,Y -105.8261,Z 120,A -69.1186,B 24.9544,C -1.5596,E1 25.0668,E2 515.0956} C_DIS
LIN {X 50.7975,Y -104.2449,Z 120,A -66.6088,B 24.9524,C -1.5935,E1 25.0733,E2 512.5121} C_DIS
LIN {X 55.0062,Y -102.0852,Z 120,A -65.2028,B 24.9548,C -1.5541,E1 25.0765,E2 511.2034} C_DIS
LIN {X 58.9017,Y -99.8879,Z 120,A -62.779,B 24.9539,C -1.568,E1 25.0824,E2 508.7537} C_DIS
LIN {X 61.4708,Y -98.3276,Z 120,A -61.3026,B 24.9538,C -1.5705,E1 25.0859,E2 507.2764} C_DIS
LIN {X 64.701,Y -96.2336,Z 120,A -59.3511,B 24.9534,C -1.5766,E1 25.0905,E2 505.3169} C_DIS
LIN {X 67.5174,Y -94.2784,Z 120,A -57.7696,B 24.9535,C -1.5748,E1 25.0941,E2 503.7451} C_DIS
LIN {X 69.9687,Y -92.4744,Z 120,A -56.0795,B 24.9528,C -1.5867,E1 25.0979,E2 502.0328} C_DIS
LIN {X 73.2767,Y -89.8756,Z 120,A -54.2005,B 24.9531,C -1.582,E1 25.102,E2 500.1722} C_DIS
LIN {X 75.4243,Y -88.0809,Z 120,A -52.684,B 24.9525,C -1.5914,E1 25.1052,E2 498.6392} C_DIS
LIN {X 78.3789,Y -85.4618,Z 120,A -50.8829,B 24.9527,C -1.589,E1 25.109,E2 496.8511} C_DIS
LIN {X 80.6243,Y -83.3471,Z 120,A -49.3444,B 24.9524,C -1.5933,E1 25.1121,E2 495.3087} C_DIS
LIN {X 83.2766,Y -80.6974,Z 120,A -47.4448,B 24.952,C -1.6001,E1 25.1158,E2 493.4011} C_DIS
LIN {X 85.6376,Y -78.1874,Z 120,A -45.6684,B 24.9516,C -1.608,E1 25.1192,E2 491.614} C_DIS
LIN {X 88.3342,Y -75.127,Z 120,A -43.8217,B 24.9517,C -1.6052,E1 25.1225,E2 489.7821} C_DIS
LIN {X 90.225,Y -72.8456,Z 120,A -42.348,B 24.9515,C -1.6096,E1 25.1252,E2 488.3049} C_DIS
LIN {X 92.4014,Y -70.0659,Z 120,A -40.4921,B 24.9508,C -1.6196,E1 25.1283,E2 486.4342} C_DIS
LIN {X 94.6574,Y -66.9862,Z 120,A -38.7495,B 24.9509,C -1.6181,E1 25.1312,E2 484.7037} C_DIS
LIN {X 96.6802,Y -64.0311,Z 120,A -36.9583,B 24.9506,C -1.6241,E1 25.134,E2 482.9071} C_DIS
LIN {X 99.5575,Y -59.4607,Z 120,A -33.5888,B 24.948,C -1.6655,E1 25.139,E2 479.4573} C_DIS
LIN {X 101.9355,Y -55.2823,Z 120,A -32.3118,B 24.9508,C -1.6199,E1 25.1406,E2 478.2944} C_DIS
LIN {X 105.487,Y -48.1643,Z 120,A -27.9163,B 24.9487,C -1.6538,E1 25.1461,E2 473.8424} C_DIS
LIN {X 107.2074,Y -44.2022,Z 120,A -26.0496,B 24.9491,C -1.6476,E1 25.1481,E2 472.0004} C_DIS
LIN {X 108.5534,Y -40.7829,Z 120,A -24.1036,B 24.9484,C -1.6595,E1 25.15,E2 470.0372} C_DIS
LIN {X 110.3421,Y -35.6596,Z 120,A -21.4117,B 24.9478,C -1.6685,E1 25.1525,E2 467.3393} C_DIS
LIN {X 111.3057,Y -32.5306,Z 120,A -19.7402,B 24.9473,C -1.6762,E1 25.1538,E2 465.6592} C_DIS
LIN {X 112.4513,Y -28.3189,Z 120,A -17.5437,B 24.9468,C -1.6851,E1 25.1554,E2 463.4545} C_DIS
LIN {X 113.3443,Y -24.497,Z 120,A -15.798,B 24.947,C -1.6821,E1 25.1564,E2 461.726} C_DIS
LIN {X 113.9721,Y -21.3922,Z 120,A -14.2619,B 24.9467,C -1.6857,E1 25.1572,E2 460.1902} C_DIS
LIN {X 114.5104,Y -18.2944,Z 120,A -12.3857,B 24.9454,C -1.7063,E1 25.1581,E2 458.2766} C_DIS
LIN {X 115.1625,Y -13.5863,Z 120,A -10.0478,B 24.945,C -1.7134,E1 25.1589,E2 455.9357} C_DIS
LIN {X 115.6023,Y -9.1155,Z 120,A -8.1437,B 24.9455,C -1.7055,E1 25.1594,E2 454.0615} C_DIS
LIN {X 115.8254,Y -5.6493,Z 120,A -6.443,B 24.9452,C -1.7104,E1 25.1596,E2 452.3595} C_DIS
LIN {X 115.9464,Y -1.868,Z 120,A -4.5605,B 24.9447,C -1.7171,E1 25.1598,E2 450.4723} C_DIS
LIN {X 115.9592,Y 0.7366,Z 120,A -3.206,B 24.9443,C -1.7246,E1 25.1598,E2 449.1083} C_DIS
LIN {X 115.8597,Y 4.8512,Z 120,A -1.235,B 24.944,C -1.7282,E1 25.1596,E2 447.1405} C_DIS
LIN {X 115.613,Y 8.9818,Z 120,A 0.8356,B 24.9435,C -1.736,E1 25.1592,E2 445.0636} C_DIS
LIN {X 115.338,Y 12.0057,Z 120,A 2.2271,B 24.9435,C -1.7357,E1 25.1588,E2 443.6812} C_DIS
LIN {X 114.9332,Y 15.4148,Z 120,A 3.8546,B 24.9435,C -1.7378,E1 25.1582,E2 442.0584} C_DIS
LIN {X 114.4957,Y 18.3878,Z 120,A 5.6418,B 24.9421,C -1.757,E1 25.1575,E2 440.2364} C_DIS
LIN {X 113.8154,Y 22.2063,Z 120,A 8.0858,B 24.94,C -1.7885,E1 25.1561,E2 437.7325} C_DIS
LIN {X 112.7106,Y 27.2645,Z 120,A 9.5782,B 24.9429,C -1.7454,E1 25.1553,E2 436.3503} C_DIS
LIN {X 112.0956,Y 29.6956,Z 120,A 11.7902,B 24.9396,C -1.7957,E1 25.1536,E2 434.0324} C_DIS
LIN {X 110.7641,Y 34.3264,Z 120,A 13.4364,B 24.9414,C -1.7678,E1 25.1523,E2 432.4613} C_DIS
LIN {X 109.6677,Y 37.6886,Z 120,A 15.3242,B 24.9406,C -1.7797,E1 25.1506,E2 430.5561} C_DIS
LIN {X 108.3857,Y 41.2256,Z 120,A 16.9729,B 24.9409,C -1.7753,E1 25.149,E2 428.927} C_DIS
LIN {X 107.2033,Y 44.2121,Z 120,A 18.7342,B 24.9401,C -1.7882,E1 25.1472,E2 427.1449} C_DIS
LIN {X 105.2005,Y 48.7839,Z 120,A 21.0796,B 24.94,C -1.7897,E1 25.1445,E2 424.8089} C_DIS
LIN {X 103.6752,Y 51.9488,Z 120,A 23.0017,B 24.939,C -1.8034,E1 25.1421,E2 422.8648} C_DIS
LIN {X 101.4883,Y 56.1012,Z 120,A 25.1582,B 24.9391,C -1.8021,E1 25.1392,E2 420.7225} C_DIS
LIN {X 99.6932,Y 59.231,Z 120,A 26.8427,B 24.9391,C -1.8023,E1 25.1369,E2 419.0462} C_DIS
LIN {X 97.7786,Y 62.3413,Z 120,A 29.1384,B 24.9372,C -1.8303,E1 25.1334,E2 416.6961} C_DIS
LIN {X 95.6055,Y 65.628,Z 120,A 30.8411,B 24.9377,C -1.8237,E1 25.1307,E2 415.0173} C_DIS
LIN {X 92.725,Y 69.6351,Z 120,A 32.9944,B 24.9382,C -1.8165,E1 25.1272,E2 412.8915} C_DIS
LIN {X 89.8362,Y 73.3253,Z 120,A 35.2677,B 24.9379,C -1.8201,E1 25.1233,E2 410.6204} C_DIS
LIN {X 87.6373,Y 75.94,Z 120,A 37.0646,B 24.9373,C -1.8291,E1 25.12,E2 408.8102} C_DIS
LIN {X 84.1497,Y 79.7874,Z 120,A 39.6651,B 24.9368,C -1.8365,E1 25.115,E2 406.2037} C_DIS
LIN {X 81.3391,Y 82.6497,Z 120,A 41.4674,B 24.9371,C -1.8325,E1 25.1115,E2 404.4186} C_DIS
LIN {X 77.5369,Y 86.2269,Z 120,A 43.8353,B 24.9374,C -1.828,E1 25.1067,E2 402.0709} C_DIS
LIN {X 75.4547,Y 88.055,Z 120,A 45.4792,B 24.9363,C -1.8434,E1 25.1032,E2 400.3972} C_DIS
LIN {X 71.1897,Y 91.5384,Z 120,A 48.2671,B 24.9357,C -1.8516,E1 25.0971,E2 397.6004} C_DIS
LIN {X 68.1237,Y 93.8422,Z 120,A 50.2552,B 24.9352,C -1.8592,E1 25.0926,E2 395.6013} C_DIS
LIN {X 65.3356,Y 95.8039,Z 120,A 51.9591,B 24.9349,C -1.8629,E1 25.0887,E2 393.8944} C_DIS
LIN {X 61.4434,Y 98.3447,Z 120,A 54.0099,B 24.9355,C -1.8553,E1 25.0839,E2 391.8683} C_DIS
LIN {X 58.1503,Y 100.328,Z 120,A 56.0258,B 24.9349,C -1.8634,E1 25.079,E2 389.8393} C_DIS
LIN {X 55.0347,Y 102.0698,Z 120,A 57.7418,B 24.9349,C -1.8637,E1 25.0748,E2 388.1277} C_DIS
LIN {X 50.3868,Y 104.4422,Z 120,A 60.4668,B 24.9342,C -1.8737,E1 25.068,E2 385.3864} C_DIS
LIN {X 46.2345,Y 106.3455,Z 120,A 62.4698,B 24.9348,C -1.8647,E1 25.063,E2 383.4095} C_DIS
LIN {X 43.0528,Y 107.675,Z 120,A 64.1312,B 24.9348,C -1.8646,E1 25.0587,E2 381.7523} C_DIS
LIN {X 39.5384,Y 109.0125,Z 120,A 65.9943,B 24.9347,C -1.8666,E1 25.0538,E2 379.8883} C_DIS
LIN {X 36.4319,Y 110.0914,Z 120,A 68.0701,B 24.9332,C -1.8883,E1 25.0482,E2 377.7652} C_DIS
LIN {X 33.2575,Y 111.0898,Z 120,A 69.5627,B 24.9336,C -1.8827,E1 25.0442,E2 376.2885} C_DIS
LIN {X 29.3249,Y 112.1929,Z 120,A 71.3636,B 24.9341,C -1.8743,E1 25.0394,E2 374.5105} C_DIS
LIN {X 23.9824,Y 113.4561,Z 120,A 73.9681,B 24.9344,C -1.8709,E1 25.0324,E2 371.9176} C_DIS
LIN {X 19.8868,Y 114.2449,Z 120,A 76.0113,B 24.9344,C -1.8709,E1 25.0268,E2 369.8766} C_DIS
LIN {X 15.8453,Y 114.8744,Z 120,A 78.363,B 24.9333,C -1.8861,E1 25.0202,E2 367.4909} C_DIS
LIN {X 10.3035,Y 115.503,Z 120,A 80.9487,B 24.9338,C -1.879,E1 25.013,E2 364.9238} C_DIS
LIN {X 6.4467,Y 115.7818,Z 120,A 82.7612,B 24.9341,C -1.8747,E1 25.008,E2 363.1222} C_DIS
LIN {X 1.9914,Y 115.9441,Z 120,A 85.2526,B 24.9332,C -1.8872,E1 25.001,E2 360.6018} C_DIS
LIN {X -2.2795,Y 115.9388,Z 120,A 87.0656,B 24.9342,C -1.8736,E1 24.996,E2 358.8209} C_DIS
LIN {X -5.127,Y 115.8478,Z 120,A 88.4957,B 24.9342,C -1.8742,E1 24.992,E2 357.3893} C_DIS
LIN {X -10.5248,Y 115.4826,Z 120,A 91.0966,B 24.9345,C -1.8698,E1 24.9848,E2 354.7975} C_DIS
LIN {X -16.2347,Y 114.8191,Z 120,A 93.6874,B 24.9353,C -1.8574,E1 24.9777,E2 352.2345} C_DIS
LIN {X -20.4506,Y 114.1436,Z 120,A 96.1618,B 24.9343,C -1.8715,E1 24.9708,E2 349.7242} C_DIS
LIN {X -28.1828,Y 112.4865,Z 120,A 99.9976,B 24.9348,C -1.8649,E1 24.9604,E2 345.8995} C_DIS
LIN {X -32.1029,Y 111.43,Z 120,A 102.1363,B 24.9346,C -1.8684,E1 24.9546,E2 343.7489} C_DIS
LIN {X -35.7648,Y 110.308,Z 120,A 103.9729,B 24.9349,C -1.8639,E1 24.9497,E2 341.9199} C_DIS
LIN {X -38.9725,Y 109.2177,Z 120,A 105.6941,B 24.9349,C -1.8637,E1 24.9452,E2 340.1957} C_DIS
LIN {X -44.0201,Y 107.2815,Z 120,A 108.1741,B 24.9357,C -1.852,E1 24.9388,E2 337.7384} C_DIS
LIN {X -48.4179,Y 105.3696,Z 120,A 111.0296,B 24.9345,C -1.869,E1 24.9314,E2 334.8354} C_DIS
LIN {X -52.8478,Y 103.2187,Z 120,A 113.3822,B 24.935,C -1.8616,E1 24.9255,E2 332.4941} C_DIS
LIN {X -56.8716,Y 101.0581,Z 120,A 115.474,B 24.9358,C -1.8507,E1 24.9204,E2 330.4223} C_DIS
LIN {X -60.094,Y 99.1752,Z 120,A 117.3085,B 24.9361,C -1.8469,E1 24.9161,E2 328.5912} C_DIS
LIN {X -63.5232,Y 97.015,Z 120,A 119.5423,B 24.9357,C -1.8528,E1 24.9108,E2 326.3362} C_DIS
LIN {X -67.4326,Y 94.3389,Z 120,A 121.5315,B 24.937,C -1.8333,E1 24.9063,E2 324.3866} C_DIS
LIN {X -70.0253,Y 92.4319,Z 120,A 123.2734,B 24.9368,C -1.8363,E1 24.9024,E2 322.6315} C_DIS
LIN {X -73.0336,Y 90.0726,Z 120,A 125.1028,B 24.9372,C -1.8297,E1 24.8984,E2 320.8109} C_DIS
LIN {X -75.7441,Y 87.8084,Z 120,A 126.9477,B 24.9372,C -1.8299,E1 24.8945,E2 318.9585} C_DIS
LIN {X -78.4841,Y 85.3653,Z 120,A 128.6457,B 24.9379,C -1.8209,E1 24.891,E2 317.275} C_DIS
LIN {X -81.0191,Y 82.9658,Z 120,A 130.5709,B 24.9376,C -1.825,E1 24.8871,E2 315.332} C_DIS
LIN {X -83.7116,Y 80.2462,Z 120,A 132.2846,B 24.9384,C -1.8131,E1 24.8838,E2 313.6394} C_DIS
LIN {X -86.9377,Y 76.7411,Z 120,A 134.8568,B 24.9382,C -1.8161,E1 24.8789,E2 311.0487} C_DIS
LIN {X -89.7251,Y 73.4624,Z 120,A 136.8579,B 24.9389,C -1.8053,E1 24.8754,E2 309.0639} C_DIS
LIN {X -92.4687,Y 69.9763,Z 120,A 139.7923,B 24.9372,C -1.8302,E1 24.8703,E2 306.0562} C_DIS
LIN {X -95.4112,Y 65.9075,Z 120,A 141.6436,B 24.9395,C -1.7972,E1 24.8674,E2 304.2745} C_DIS
LIN {X -97.5388,Y 62.715,Z 120,A 143.4327,B 24.9401,C -1.7874,E1 24.8647,E2 302.4997} C_DIS
LIN {X -101.2236,Y 56.5753,Z 120,A 146.936,B 24.9409,C -1.7757,E1 24.8598,E2 299.0062} C_DIS
LIN {X -102.9336,Y 53.4056,Z 120,A 148.7356,B 24.9412,C -1.7712,E1 24.8574,E2 297.2078} C_DIS
LIN {X -104.9259,Y 49.3738,Z 120,A 150.9489,B 24.9417,C -1.7641,E1 24.8547,E2 294.9994} C_DIS
LIN {X -106.5372,Y 45.7925,Z 120,A 153.1727,B 24.9413,C -1.7698,E1 24.8522,E2 292.7497} C_DIS
LIN {X -108.0021,Y 42.2204,Z 120,A 154.84,B 24.9423,C -1.7541,E1 24.8505,E2 291.1107} C_DIS
LIN {X -109.216,Y 38.9772,Z 120,A 157.2378,B 24.9408,C -1.7768,E1 24.8481,E2 288.645} C_DIS
LIN {X -110.6063,Y 34.8352,Z 120,A 158.6544,B 24.9433,C -1.7396,E1 24.847,E2 287.309} C_DIS
LIN {X -111.8807,Y 30.4918,Z 120,A 161.7546,B 24.9414,C -1.7679,E1 24.8446,E2 284.1234} C_DIS
LIN {X -113.0452,Y 25.8418,Z 120,A 163.6654,B 24.9432,C -1.7414,E1 24.8434,E2 282.2645} C_DIS
LIN {X -113.784,Y 22.3695,Z 120,A 165.2718,B 24.9439,C -1.7297,E1 24.8425,E2 280.6766} C_DIS
LIN {X -114.9655,Y 15.1656,Z 120,A 169.8204,B 24.9422,C -1.7567,E1 24.8407,E2 276.0365} C_DIS
LIN {X -115.5988,Y 9.1595,Z 120,A 171.4558,B 24.9464,C -1.6917,E1 24.8403,E2 274.5462} C_DIS
LIN {X -115.8568,Y 4.9168,Z 120,A 173.933,B 24.9458,C -1.7001,E1 24.8399,E2 272.0341} C_DIS
LIN {X -115.9615,Y -0.3031,Z 120,A 176.3505,B 24.9468,C -1.6851,E1 24.8399,E2 269.6379} C_DIS
LIN {X -115.9189,Y -3.1546,Z 120,A 178.6719,B 24.9447,C -1.7179,E1 24.8399,E2 267.2243} C_DIS
LIN {X -115.6921,Y -7.8949,Z 120,A -179.7688,B 24.9472,C -1.678,E1 24.8402,E2 265.7506} C_DIS
LIN {X -115.1937,Y -13.3199,Z 120,A -177.2557,B 24.9482,C -1.6621,E1 24.8409,E2 263.2605} C_DIS
LIN {X -114.1478,Y -20.427,Z 120,A -173.3633,B 24.9481,C -1.6647,E1 24.8425,E2 259.3387} C_DIS
LIN {X -113.528,Y -23.632,Z 120,A -171.6861,B 24.9482,C -1.6622,E1 24.8435,E2 257.6574} C_DIS
LIN {X -112.6727,Y -27.4196,Z 120,A -169.8788,B 24.9489,C -1.6517,E1 24.8446,E2 255.8647} C_DIS
LIN {X -111.9001,Y -30.4202,Z 120,A -168.2022,B 24.9489,C -1.6529,E1 24.8458,E2 254.1754} C_DIS
LIN {X -110.7865,Y -34.2541,Z 120,A -166.2526,B 24.9492,C -1.646,E1 24.8474,E2 252.2311} C_DIS
LIN {X -109.3038,Y -38.7271,Z 120,A -164.0458,B 24.95,C -1.6339,E1 24.8493,E2 250.0404} C_DIS
LIN {X -108.2863,Y -41.4881,Z 120,A -162.3947,B 24.9497,C -1.6377,E1 24.851,E2 248.3709} C_DIS
LIN {X -106.3232,Y -46.2855,Z 120,A -159.8668,B 24.9503,C -1.6289,E1 24.8537,E2 245.8501} C_DIS
LIN {X -104.8269,Y -49.5863,Z 120,A -157.9834,B 24.9503,C -1.6276,E1 24.8559,E2 243.9595} C_DIS
LIN {X -103.0451,Y -53.1875,Z 120,A -155.926,B 24.9505,C -1.6251,E1 24.8585,E2 241.8972} C_DIS
LIN {X -101.197,Y -56.623,Z 120,A -154.1935,B 24.9513,C -1.6117,E1 24.8608,E2 240.1874} C_DIS
LIN {X -99.4404,Y -59.6576,Z 120,A -152.1987,B 24.951,C -1.6179,E1 24.8637,E2 238.1674} C_DIS
LIN {X -96.7243,Y -63.9642,Z 120,A -149.9738,B 24.9521,C -1.5992,E1 24.867,E2 235.9759} C_DIS
LIN {X -94.8859,Y -66.6632,Z 120,A -148.1751,B 24.9519,C -1.6028,E1 24.8699,E2 234.1597} C_DIS
LIN {X -90.3172,Y -72.7319,Z 120,A -144.67,B 24.953,C -1.5832,E1 24.8758,E2 230.6847} C_DIS
LIN {X -88.5158,Y -74.9138,Z 120,A -142.8387,B 24.9521,C -1.5981,E1 24.8792,E2 228.8094} C_DIS
LIN {X -85.4178,Y -78.4269,Z 120,A -140.7557,B 24.953,C -1.5831,E1 24.883,E2 226.7529} C_DIS
LIN {X -82.8657,Y -81.1205,Z 120,A -137.9052,B 24.9507,C -1.6224,E1 24.8888,E2 223.7966} C_DIS
LIN {X -78.4017,Y -85.441,Z 120,A -136.099,B 24.9543,C -1.5622,E1 24.8922,E2 222.1263} C_DIS
LIN {X -76.8116,Y -86.8753,Z 120,A -134.3165,B 24.9526,C -1.5908,E1 24.8961,E2 220.2686} C_DIS
LIN {X -74.0167,Y -89.2666,Z 120,A -132.9673,B 24.954,C -1.5674,E1 24.8989,E2 218.97} C_DIS
LIN {X -70.9904,Y -91.692,Z 120,A -130.9517,B 24.954,C -1.5681,E1 24.9033,E2 216.9452} C_DIS
LIN {X -68.4124,Y -93.6308,Z 120,A -129.567,B 24.9546,C -1.5564,E1 24.9064,E2 215.5835} C_DIS
LIN {X -65.7573,Y -95.5156,Z 120,A -127.8086,B 24.9544,C -1.5601,E1 24.9104,E2 213.8103} C_DIS
LIN {X -62.6321,Y -97.592,Z 120,A -125.9584,B 24.9546,C -1.557,E1 24.9147,E2 211.9615} C_DIS
LIN {X -58.5975,Y -100.0676,Z 120,A -123.7182,B 24.955,C -1.5492,E1 24.9201,E2 209.7328} C_DIS
LIN {X -55.9629,Y -101.5656,Z 120,A -121.8644,B 24.9543,C -1.5625,E1 24.9247,E2 207.8421} C_DIS
LIN {X -52.8337,Y -103.2259,Z 120,A -120.1734,B 24.9545,C -1.5577,E1 24.9289,E2 206.1579} C_DIS
LIN {X -48.913,Y -105.1404,Z 120,A -118.1918,B 24.9551,C -1.5476,E1 24.9338,E2 204.1953} C_DIS
LIN {X -45.6405,Y -106.6037,Z 120,A -116.1107,B 24.9545,C -1.5591,E1 24.9392,E2 202.0818} C_DIS
LIN {X -40.8732,Y -108.5191,Z 120,A -113.8763,B 24.9554,C -1.5434,E1 24.945,E2 199.88} C_DIS
LIN {X -35.9176,Y -110.2586,Z 120,A -111.0694,B 24.955,C -1.5505,E1 24.9524,E2 197.051} C_DIS
LIN {X -32.627,Y -111.2771,Z 120,A -109.6148,B 24.9557,C -1.5384,E1 24.9563,E2 195.6226} C_DIS
LIN {X -28.047,Y -112.5197,Z 120,A -107.3364,B 24.9559,C -1.534,E1 24.9624,E2 193.3512} C_DIS
LIN {X -23.7663,Y -113.5004,Z 120,A -105.2246,B 24.9561,C -1.5304,E1 24.9681,E2 191.2453} C_DIS
LIN {X -19.4295,Y -114.3222,Z 120,A -102.6276,B 24.9551,C -1.5481,E1 24.9754,E2 188.6037} C_DIS
LIN {X -14.1061,Y -115.1016,Z 120,A -100.0683,B 24.9554,C -1.5431,E1 24.9824,E2 186.0543} C_DIS
LIN {X -10.4067,Y -115.4935,Z 120,A -98.4119,B 24.9559,C -1.5348,E1 24.987,E2 184.4165} C_DIS
LIN {X -7.0564,Y -115.748,Z 120,A -96.5669,B 24.9554,C -1.5431,E1 24.9922,E2 182.5513} C_DIS
LIN {X -2.6351,Y -115.9322,Z 120,A -94.6772,B 24.9561,C -1.5301,E1 24.9974,E2 180.692} C_DIS
LIN {X 0.827,Y -115.9579,Z 120,A -93.4935,B 24.9575,C -1.507,E1 25.0005,E2 179.5631} C_DIS
Enddeposition()
LIN {X 0.827,Y -115.9579,Z 120,A -93.4935,B 24.9575,C -1.507,E1 25.0005,E2 179.5631} C_DIS
Startdeposition()
$VEL.CP = VEL_PRINT
LIN {X -0.7761,Y -115.0723,Z 120,A -94.7898,B 24.9578,C -1.5006,E1 24.9969,E2 180.8745} C_DIS
LIN {X -4.2948,Y -114.9963,Z 120,A -96.5151,B 24.9578,C -1.5016,E1 24.9921,E2 182.5979} C_DIS
LIN {X -7.4975,Y -114.8307,Z 120,A -97.7633,B 24.9569,C -1.5167,E1 24.9887,E2 183.8107} C_DIS
LIN {X -10.9426,Y -114.554,Z 120,A -99.545,B 24.957,C -1.5141,E1 24.9837,E2 185.5993} C_DIS
LIN {X -15.866,Y -113.9763,Z 120,A -102.3922,B 24.9579,C -1.4982,E1 24.9757,E2 188.4863} C_DIS
LIN {X -19.5938,Y -113.3962,Z 120,A -103.9076,B 24.957,C -1.5144,E1 24.9716,E2 189.9647} C_DIS
LIN {X -22.2002,Y -112.914,Z 120,A -105.3959,B 24.9574,C -1.5077,E1 24.9675,E2 191.4706} C_DIS
LIN {X -26.2007,Y -112.0529,Z 120,A -107.5716,B 24.9577,C -1.5028,E1 24.9616,E2 193.6608} C_DIS
LIN {X -29.5601,Y -111.2144,Z 120,A -108.7813,B 24.9564,C -1.5258,E1 24.9584,E2 194.8176} C_DIS
LIN {X -32.6279,Y -110.3524,Z 120,A -110.3916,B 24.9564,C -1.5258,E1 24.9541,E2 196.4303} C_DIS
LIN {X -38.1649,Y -108.5618,Z 120,A -113.3925,B 24.9564,C -1.5238,E1 24.9461,E2 199.4419} C_DIS
LIN {X -41.6779,Y -107.263,Z 120,A -115.934,B 24.958,C -1.4969,E1 24.9393,E2 202.0525} C_DIS
LIN {X -45.9357,Y -105.509,Z 120,A -117.5841,B 24.9563,C -1.5265,E1 24.9352,E2 203.6362} C_DIS
LIN {X -49.5019,Y -103.8842,Z 120,A -119.4168,B 24.9559,C -1.5337,E1 24.9306,E2 205.4563} C_DIS
LIN {X -53.0144,Y -102.138,Z 120,A -121.7146,B 24.9566,C -1.5217,E1 24.9248,E2 207.7889} C_DIS
LIN {X -56.9568,Y -99.9917,Z 120,A -123.534,B 24.9554,C -1.5422,E1 24.9205,E2 209.5647} C_DIS
LIN {X -61.5892,Y -97.2083,Z 120,A -126.4858,B 24.9558,C -1.5353,E1 24.9134,E2 212.5421} C_DIS
LIN {X -65.039,Y -94.9341,Z 120,A -128.4533,B 24.9554,C -1.5424,E1 24.9088,E2 214.4993} C_DIS
LIN {X -68.3224,Y -92.5983,Z 120,A -130.567,B 24.9554,C -1.5414,E1 24.904,E2 216.6228} C_DIS
LIN {X -71.3668,Y -90.2718,Z 120,A -132.4143,B 24.9551,C -1.5473,E1 24.9,E2 218.4626} C_DIS
LIN {X -73.2386,Y -88.7609,Z 120,A -134.0089,B 24.956,C -1.5332,E1 24.8965,E2 220.0969} C_DIS
LIN {X -75.8157,Y -86.5692,Z 120,A -135.3299,B 24.9549,C -1.5515,E1 24.8938,E2 221.3796} C_DIS
LIN {X -78.1664,Y -84.454,Z 120,A -137.7331,B 24.9567,C -1.5208,E1 24.8887,E2 223.8656} C_DIS
LIN {X -82.0228,Y -80.7127,Z 120,A -139.5475,B 24.9543,C -1.5616,E1 24.8853,E2 225.5905} C_DIS
LIN {X -84.5376,Y -78.0753,Z 120,A -141.3961,B 24.9542,C -1.5642,E1 24.8817,E2 227.4409} C_DIS
LIN {X -87.3877,Y -74.8714,Z 120,A -143.5381,B 24.9539,C -1.5689,E1 24.8778,E2 229.5816} C_DIS
LIN {X -89.7533,Y -72.02,Z 120,A -146.1915,B 24.9555,C -1.5405,E1 24.873,E2 232.3149} C_DIS
LIN {X -92.8638,Y -67.9598,Z 120,A -147.8867,B 24.9532,C -1.5812,E1 24.8703,E2 233.9212} C_DIS
LIN {X -94.7434,Y -65.3155,Z 120,A -149.6852,B 24.9534,C -1.5779,E1 24.8674,E2 235.7367} C_DIS
LIN {X -97.9147,Y -60.4571,Z 120,A -152.546,B 24.9528,C -1.5866,E1 24.8631,E2 238.5912} C_DIS
LIN {X -99.8552,Y -57.1943,Z 120,A -154.1986,B 24.952,C -1.6013,E1 24.8608,E2 240.2173} C_DIS
LIN {X -101.7578,Y -53.7364,Z 120,A -156.4231,B 24.9523,C -1.5962,E1 24.8578,E2 242.4656} C_DIS
LIN {X -103.5771,Y -50.141,Z 120,A -158.1548,B 24.9513,C -1.6129,E1 24.8557,E2 244.1668} C_DIS
LIN {X -104.6764,Y -47.806,Z 120,A -160.1612,B 24.9528,C -1.5876,E1 24.8533,E2 246.2445} C_DIS
LIN {X -106.1785,Y -44.3675,Z 120,A -161.6622,B 24.9516,C -1.6077,E1 24.8517,E2 247.7059} C_DIS
LIN {X -107.8313,Y -40.1872,Z 120,A -164.3817,B 24.9523,C -1.5952,E1 24.8489,E2 250.4707} C_DIS
LIN {X -109.2196,Y -36.2438,Z 120,A -166.0199,B 24.9509,C -1.6191,E1 24.8475,E2 252.0613} C_DIS
LIN {X -110.3177,Y -32.7451,Z 120,A -167.7476,B 24.9503,C -1.6286,E1 24.8461,E2 253.7762} C_DIS
LIN {X -111.2844,Y -29.2996,Z 120,A -169.5577,B 24.95,C -1.6329,E1 24.8448,E2 255.5865} C_DIS
LIN {X -112.1655,Y -25.7129,Z 120,A -171.4146,B 24.9497,C -1.6379,E1 24.8436,E2 257.4422} C_DIS
LIN {X -112.9548,Y -21.9887,Z 120,A -173.3442,B 24.9494,C -1.6425,E1 24.8425,E2 259.3723} C_DIS
LIN {X -114.0497,Y -15.336,Z 120,A -176.7046,B 24.9488,C -1.653,E1 24.8411,E2 262.7276} C_DIS
LIN {X -114.7296,Y -8.9114,Z 120,A 179.2687,B 24.9501,C -1.6315,E1 24.84,E2 266.83} C_DIS
LIN {X -115.0165,Y -3.6671,Z 120,A 177.4798,B 24.9476,C -1.6725,E1 24.8398,E2 268.5319} C_DIS
LIN {X -115.0408,Y 2.874,Z 120,A 173.6531,B 24.9483,C -1.6605,E1 24.8399,E2 272.4101} C_DIS
LIN {X -114.8772,Y 6.7547,Z 120,A 172.2346,B 24.9467,C -1.6872,E1 24.8401,E2 273.7735} C_DIS
LIN {X -114.6155,Y 10.2766,Z 120,A 169.821,B 24.9479,C -1.6671,E1 24.8407,E2 276.2496} C_DIS
LIN {X -114.1342,Y 14.6836,Z 120,A 168.4686,B 24.9453,C -1.708,E1 24.8412,E2 277.5125} C_DIS
LIN {X -113.406,Y 19.5349,Z 120,A 165.7532,B 24.9455,C -1.7051,E1 24.8423,E2 280.2511} C_DIS
LIN {X -112.7668,Y 22.9331,Z 120,A 164.0415,B 24.9451,C -1.711,E1 24.8432,E2 281.9587} C_DIS
LIN {X -111.0856,Y 30.0369,Z 120,A 160.4042,B 24.9444,C -1.7226,E1 24.8457,E2 285.5897} C_DIS
LIN {X -110.1101,Y 33.443,Z 120,A 158.6779,B 24.9439,C -1.7296,E1 24.847,E2 287.3092} C_DIS
LIN {X -107.6332,Y 40.7101,Z 120,A 154.875,B 24.9431,C -1.7424,E1 24.8505,E2 291.1033} C_DIS
LIN {X -105.0064,Y 47.0736,Z 120,A 151.3386,B 24.9427,C -1.7486,E1 24.8543,E2 294.6446} C_DIS
LIN {X -102.8623,Y 51.5933,Z 120,A 148.8448,B 24.9422,C -1.7559,E1 24.8573,E2 297.1344} C_DIS
LIN {X -100.766,Y 55.577,Z 120,A 146.6429,B 24.9417,C -1.7641,E1 24.8602,E2 299.3283} C_DIS
LIN {X -96.5301,Y 62.6458,Z 120,A 142.4697,B 24.9411,C -1.7731,E1 24.8662,E2 303.5016} C_DIS
LIN {X -93.965,Y 66.4308,Z 120,A 139.8491,B 24.9416,C -1.7657,E1 24.8704,E2 306.1528} C_DIS
LIN {X -89.8065,Y 71.9543,Z 120,A 136.5454,B 24.9406,C -1.7805,E1 24.876,E2 309.4368} C_DIS
LIN {X -87.4578,Y 74.789,Z 120,A 135.0164,B 24.9394,C -1.7976,E1 24.8787,E2 310.9323} C_DIS
LIN {X -84.4078,Y 78.2168,Z 120,A 132.3944,B 24.94,C -1.7898,E1 24.8837,E2 313.5846} C_DIS
LIN {X -81.6361,Y 81.1042,Z 120,A 130.5383,B 24.9393,C -1.8002,E1 24.8872,E2 315.4237} C_DIS
LIN {X -78.9109,Y 83.7574,Z 120,A 128.6247,B 24.939,C -1.804,E1 24.8911,E2 317.3364} C_DIS
LIN {X -76.4531,Y 86.0076,Z 120,A 126.9746,B 24.9387,C -1.8082,E1 24.8945,E2 318.9831} C_DIS
LIN {X -73.1638,Y 88.823,Z 120,A 124.6989,B 24.9387,C -1.8082,E1 24.8994,E2 321.2676} C_DIS
LIN {X -70.1285,Y 91.2373,Z 120,A 122.8537,B 24.9382,C -1.8158,E1 24.9034,E2 323.1013} C_DIS
LIN {X -68.0277,Y 92.8141,Z 120,A 121.259,B 24.9388,C -1.8069,E1 24.9071,E2 324.7229} C_DIS
LIN {X -61.9983,Y 96.9457,Z 120,A 117.8658,B 24.9376,C -1.8241,E1 24.9149,E2 328.0865} C_DIS
LIN {X -58.8494,Y 98.8893,Z 120,A 116.2036,B 24.9369,C -1.8349,E1 24.9188,E2 329.7281} C_DIS
LIN {X -56.469,Y 100.2679,Z 120,A 114.3708,B 24.938,C -1.8184,E1 24.9233,E2 331.6056} C_DIS
LIN {X -52.4226,Y 102.4407,Z 120,A 112.3147,B 24.9371,C -1.8317,E1 24.9283,E2 333.6357} C_DIS
LIN {X -45.6609,Y 105.6287,Z 120,A 108.8544,B 24.936,C -1.8483,E1 24.937,E2 337.0653} C_DIS
LIN {X -39.9934,Y 107.9032,Z 120,A 105.4709,B 24.9367,C -1.8381,E1 24.9459,E2 340.4802} C_DIS
LIN {X -36.5724,Y 109.1088,Z 120,A 103.6835,B 24.9365,C -1.8412,E1 24.9506,E2 342.2638} C_DIS
LIN {X -33.1787,Y 110.189,Z 120,A 101.8826,B 24.9364,C -1.842,E1 24.9554,E2 344.0658} C_DIS
LIN {X -29.9938,Y 111.0972,Z 120,A 100.3438,B 24.936,C -1.8484,E1 24.9595,E2 345.5919} C_DIS
LIN {X -23.8195,Y 112.5848,Z 120,A 96.5542,B 24.9376,C -1.8251,E1 24.97,E2 349.4418} C_DIS
LIN {X -19.6138,Y 113.3929,Z 120,A 95.0808,B 24.9355,C -1.8543,E1 24.9739,E2 350.8473} C_DIS
LIN {X -11.9904,Y 114.4485,Z 120,A 91.5494,B 24.9345,C -1.8694,E1 24.9836,E2 354.3454} C_DIS
LIN {X -5.9718,Y 114.9204,Z 120,A 88.129,B 24.9356,C -1.853,E1 24.9932,E2 357.8062} C_DIS
LIN {X -0.5121,Y 115.0739,Z 120,A 85.4874,B 24.9354,C -1.8571,E1 25.0005,E2 360.4385} C_DIS
LIN {X 5.143,Y 114.9601,Z 120,A 82.5968,B 24.9356,C -1.8542,E1 25.0086,E2 363.3354} C_DIS
LIN {X 8.6589,Y 114.7498,Z 120,A 80.418,B 24.9368,C -1.8359,E1 25.0148,E2 365.5564} C_DIS
LIN {X 12.2903,Y 114.4171,Z 120,A 78.4583,B 24.9373,C -1.8295,E1 25.0203,E2 367.5301} C_DIS
LIN {X 16.6069,Y 113.8711,Z 120,A 76.9232,B 24.9354,C -1.856,E1 25.0244,E2 369.0008} C_DIS
LIN {X 20.4428,Y 113.2445,Z 120,A 74.8412,B 24.9359,C -1.849,E1 25.0301,E2 371.0973} C_DIS
LIN {X 23.2376,Y 112.7043,Z 120,A 73.179,B 24.9367,C -1.8377,E1 25.0347,E2 372.7841} C_DIS
LIN {X 26.588,Y 111.9634,Z 120,A 71.7132,B 24.936,C -1.8473,E1 25.0387,E2 374.2253} C_DIS
LIN {X 30.4634,Y 110.9704,Z 120,A 70.0438,B 24.9351,C -1.8601,E1 25.0431,E2 375.8617} C_DIS
LIN {X 35.4892,Y 109.4657,Z 120,A 67.2349,B 24.9359,C -1.8495,E1 25.0506,E2 378.6907} C_DIS
LIN {X 38.797,Y 108.3396,Z 120,A 64.9928,B 24.9375,C -1.8259,E1 25.0567,E2 380.9841} C_DIS
LIN {X 42.4017,Y 106.9787,Z 120,A 63.5211,B 24.9363,C -1.8436,E1 25.0604,E2 382.4107} C_DIS
LIN {X 45.4961,Y 105.7006,Z 120,A 62.0078,B 24.9359,C -1.8485,E1 25.0642,E2 383.9087} C_DIS
LIN {X 49.0505,Y 104.0988,Z 120,A 60.0903,B 24.936,C -1.8473,E1 25.0691,E2 385.8243} C_DIS
LIN {X 52.2456,Y 102.5312,Z 120,A 58.2437,B 24.9364,C -1.8418,E1 25.0737,E2 387.6791} C_DIS
LIN {X 54.8831,Y 101.1438,Z 120,A 56.81,B 24.9364,C -1.842,E1 25.0773,E2 389.1083} C_DIS
LIN {X 58.0488,Y 99.3625,Z 120,A 54.8642,B 24.937,C -1.8332,E1 25.082,E2 391.0688} C_DIS
LIN {X 61.0102,Y 97.5704,Z 120,A 53.276,B 24.9368,C -1.8366,E1 25.0858,E2 392.644} C_DIS
LIN {X 64.1484,Y 95.5375,Z 120,A 51.4465,B 24.9368,C -1.8351,E1 25.09,E2 394.4712} C_DIS
LIN {X 67.2786,Y 93.3601,Z 120,A 49.3442,B 24.9377,C -1.8227,E1 25.0949,E2 396.5955} C_DIS
LIN {X 70.4069,Y 91.0228,Z 120,A 46.6628,B 24.9402,C -1.7862,E1 25.101,E2 399.3531} C_DIS
LIN {X 74.7198,Y 87.5168,Z 120,A 45.2131,B 24.9365,C -1.8401,E1 25.1038,E2 400.6701} C_DIS
LIN {X 79.131,Y 83.5504,Z 120,A 41.7529,B 24.9385,C -1.811,E1 25.1111,E2 404.1851} C_DIS
LIN {X 81.8964,Y 80.8406,Z 120,A 39.9353,B 24.9385,C -1.8118,E1 25.1146,E2 405.993} C_DIS
LIN {X 86.5814,Y 75.8017,Z 120,A 36.5291,B 24.9389,C -1.805,E1 25.1211,E2 409.4004} C_DIS
LIN {X 90.4555,Y 71.1344,Z 120,A 33.4416,B 24.9396,C -1.7946,E1 25.1266,E2 412.498} C_DIS
LIN {X 92.7171,Y 68.1602,Z 120,A 31.9202,B 24.9389,C -1.8056,E1 25.129,E2 413.9863} C_DIS
LIN {X 94.9145,Y 65.0684,Z 120,A 29.8566,B 24.9398,C -1.7927,E1 25.1324,E2 416.0703} C_DIS
LIN {X 97.0834,Y 61.7838,Z 120,A 27.8736,B 24.9402,C -1.7865,E1 25.1354,E2 418.0579} C_DIS
LIN {X 98.9892,Y 58.6804,Z 120,A 26.0282,B 24.9406,C -1.7802,E1 25.1381,E2 419.9089} C_DIS
LIN {X 100.7358,Y 55.6312,Z 120,A 24.178,B 24.9412,C -1.7707,E1 25.1406,E2 421.7717} C_DIS
LIN {X 102.1241,Y 53.0408,Z 120,A 22.41,B 24.9424,C -1.7526,E1 25.143,E2 423.5731} C_DIS
LIN {X 103.6624,Y 49.9635,Z 120,A 21.4438,B 24.9405,C -1.7822,E1 25.1441,E2 424.4642} C_DIS
LIN {X 105.4797,Y 46.0029,Z 120,A 18.9377,B 24.9419,C -1.7603,E1 25.147,E2 427.0084} C_DIS
LIN {X 106.8848,Y 42.6408,Z 120,A 17.0797,B 24.9424,C -1.753,E1 25.149,E2 428.8735} C_DIS
LIN {X 108.1836,Y 39.2247,Z 120,A 15.3031,B 24.9426,C -1.7496,E1 25.1507,E2 430.6483} C_DIS
LIN {X 109.3164,Y 35.9507,Z 120,A 13.5627,B 24.943,C -1.7436,E1 25.1522,E2 432.3928} C_DIS
LIN {X 111.1921,Y 29.6428,Z 120,A 10.2917,B 24.9437,C -1.7338,E1 25.1548,E2 435.6682} C_DIS
LIN {X 112.4973,Y 24.2211,Z 120,A 7.4302,B 24.9445,C -1.7212,E1 25.1566,E2 438.5429} C_DIS
LIN {X 113.735,Y 17.5092,Z 120,A 4.2611,B 24.9445,C -1.7211,E1 25.1581,E2 441.6936} C_DIS
LIN {X 114.2087,Y 14.1089,Z 120,A 2.4815,B 24.9451,C -1.7123,E1 25.1587,E2 443.4834} C_DIS
LIN {X 114.7111,Y 9.1421,Z 120,A -0.2242,B 24.9462,C -1.6941,E1 25.1594,E2 446.2161} C_DIS
LIN {X 115.0039,Y 4.0773,Z 120,A -2.4604,B 24.9459,C -1.6994,E1 25.1597,E2 448.4266} C_DIS
LIN {X 115.0712,Y 1.0001,Z 120,A -4.2153,B 24.9469,C -1.684,E1 25.1597,E2 450.2072} C_DIS
LIN {X 114.9541,Y -5.2827,Z 120,A -7.1639,B 24.9469,C -1.6822,E1 25.1595,E2 453.1425} C_DIS
LIN {X 114.6588,Y -9.7972,Z 120,A -9.8185,B 24.9486,C -1.6561,E1 25.159,E2 455.8429} C_DIS
LIN {X 114.2464,Y -13.7892,Z 120,A -11.182,B 24.9472,C -1.6792,E1 25.1585,E2 457.1438} C_DIS
LIN {X 113.4432,Y -19.3127,Z 120,A -14.1257,B 24.9482,C -1.6624,E1 25.1573,E2 460.1099} C_DIS
LIN {X 112.566,Y -23.9065,Z 120,A -16.2773,B 24.9482,C -1.6631,E1 25.1561,E2 462.2471} C_DIS
LIN {X 112.0866,Y -26.0545,Z 120,A -17.5702,B 24.949,C -1.6504,E1 25.1553,E2 463.5626} C_DIS
LIN {X 111.0952,Y -30.0014,Z 120,A -19.4483,B 24.949,C -1.6508,E1 25.154,E2 465.4288} C_DIS
LIN {X 110.1102,Y -33.441,Z 120,A -21.2297,B 24.9493,C -1.6451,E1 25.1526,E2 467.2135} C_DIS
LIN {X 108.3602,Y -38.7395,Z 120,A -24.1015,B 24.9501,C -1.632,E1 25.15,E2 470.1001} C_DIS
LIN {X 107.0704,Y -42.1682,Z 120,A -25.7419,B 24.9499,C -1.6349,E1 25.1484,E2 471.7246} C_DIS
LIN {X 105.1635,Y -46.7251,Z 120,A -28.1197,B 24.9501,C -1.6311,E1 25.1458,E2 474.0982} C_DIS
LIN {X 102.6544,Y -52.0044,Z 120,A -31.1507,B 24.951,C -1.6166,E1 25.1421,E2 477.1472} C_DIS
LIN {X 101.1196,Y -54.9277,Z 120,A -33.1184,B 24.9522,C -1.5967,E1 25.1394,E2 479.1515} C_DIS
LIN {X 99.4218,Y -57.9484,Z 120,A -35.1362,B 24.9533,C -1.5781,E1 25.1365,E2 481.2029} C_DIS
LIN {X 97.0282,Y -61.8699,Z 120,A -36.7695,B 24.9519,C -1.6018,E1 25.1342,E2 482.7719} C_DIS
LIN {X 95.2453,Y -64.5799,Z 120,A -38.3716,B 24.9522,C -1.5978,E1 25.1317,E2 484.3754} C_DIS
LIN {X 93.078,Y -67.6673,Z 120,A -40.2983,B 24.9526,C -1.5903,E1 25.1285,E2 486.3104} C_DIS
LIN {X 90.6191,Y -70.9274,Z 120,A -42.3347,B 24.953,C -1.5846,E1 25.1251,E2 488.3507} C_DIS
LIN {X 88.3483,Y -73.7351,Z 120,A -44.0565,B 24.953,C -1.5834,E1 25.122,E2 490.0674} C_DIS
LIN {X 85.739,Y -76.7531,Z 120,A -45.9971,B 24.9532,C -1.5803,E1 25.1185,E2 492.0065} C_DIS
LIN {X 83.0623,Y -79.6428,Z 120,A -47.8473,B 24.9532,C -1.5805,E1 25.1149,E2 493.8482} C_DIS
LIN {X 80.6762,Y -82.0588,Z 120,A -49.613,B 24.9536,C -1.5729,E1 25.1114,E2 495.6245} C_DIS
LIN {X 77.7488,Y -84.8372,Z 120,A -51.5905,B 24.9538,C -1.5695,E1 25.1074,E2 497.6017} C_DIS
LIN {X 75.0535,Y -87.2325,Z 120,A -53.5196,B 24.9545,C -1.5592,E1 25.1033,E2 499.5476} C_DIS
LIN {X 71.7708,Y -89.9526,Z 120,A -55.5599,B 24.9545,C -1.5582,E1 25.0989,E2 501.5825} C_DIS
LIN {X 68.5118,Y -92.4597,Z 120,A -57.6701,B 24.9549,C -1.5509,E1 25.0942,E2 503.7022} C_DIS
LIN {X 65.2685,Y -94.7761,Z 120,A -59.6412,B 24.9551,C -1.5475,E1 25.0897,E2 505.6747} C_DIS
LIN {X 62.2675,Y -96.7729,Z 120,A -61.2233,B 24.9548,C -1.5536,E1 25.086,E2 507.237} C_DIS
LIN {X 60.0301,Y -98.1769,Z 120,A -62.6475,B 24.9552,C -1.5461,E1 25.0826,E2 508.6745} C_DIS
LIN {X 57.2693,Y -99.8121,Z 120,A -64.2084,B 24.9552,C -1.5449,E1 25.0789,E2 510.2335} C_DIS
LIN {X 52.2809,Y -102.5131,Z 120,A -67.4912,B 24.9568,C -1.5193,E1 25.0706,E2 513.5677} C_DIS
LIN {X 48.9388,Y -104.1508,Z 120,A -68.698,B 24.9553,C -1.5455,E1 25.0678,E2 514.7094} C_DIS
LIN {X 43.9186,Y -106.3659,Z 120,A -71.8177,B 24.9565,C -1.5238,E1 25.0597,E2 517.8728} C_DIS
LIN {X 39.8661,Y -107.9497,Z 120,A -73.8785,B 24.9564,C -1.5256,E1 25.0543,E2 519.9251} C_DIS
LIN {X 36.3386,Y -109.1876,Z 120,A -75.7347,B 24.9565,C -1.5234,E1 25.0494,E2 521.7826} C_DIS
LIN {X 33.5196,Y -110.0864,Z 120,A -77.6989,B 24.9579,C -1.4998,E1 25.044,E2 523.7993} C_DIS
LIN {X 29.3076,Y -111.2823,Z 120,A -79.3602,B 24.9567,C -1.5205,E1 25.0397,E2 525.4089} C_DIS
LIN {X 26.0735,Y -112.0822,Z 120,A -81.5883,B 24.9582,C -1.4937,E1 25.0334,E2 527.6973} C_DIS
LIN {X 21.5613,Y -113.0371,Z 120,A -82.7521,B 24.9555,C -1.542,E1 25.0306,E2 528.7454} C_DIS
LIN {X 16.0878,Y -113.9448,Z 120,A -85.9842,B 24.9568,C -1.5189,E1 25.0215,E2 532.029} C_DIS
LIN {X 13.0165,Y -114.3369,Z 120,A -88.1085,B 24.9583,C -1.4923,E1 25.0155,E2 534.2147} C_DIS
LIN {X 8.7219,Y -114.7447,Z 120,A -89.5572,B 24.9566,C -1.5219,E1 25.0116,E2 535.5924} C_DIS
LIN {X 3.624,Y -115.0178,Z 120,A -92.1317,B 24.9567,C -1.5195,E1 25.0044,E2 538.1719} C_DIS
LIN {X 0.8161,Y -115.0706,Z 120,A -92.9501,B 24.9553,C -1.5447,E1 25.0023,E2 538.9303} C_DIS
Enddeposition()
LIN {X 0.8161,Y -115.0706,Z 120,A -92.9501,B 24.9553,C -1.5447,E1 25.0023,E2 538.9303} C_DIS
Startdeposition()
$VEL.CP = VEL_PRINT
LIN {X 1.1447,Y -114.1837,Z 120,A -92.694,B 24.9542,C -1.564,E1 25.0032,E2 538.6284} C_DIS
LIN {X 8.5017,Y -113.8733,Z 120,A -89.1228,B 24.9544,C -1.5599,E1 25.0131,E2 535.0682} C_DIS
LIN {X 14.6979,Y -113.2387,Z 120,A -86.2843,B 24.955,C -1.549,E1 25.0209,E2 532.2576} C_DIS
LIN {X 17.9899,Y -112.7635,Z 120,A -83.9655,B 24.9533,C -1.5791,E1 25.0275,E2 529.8695} C_DIS
LIN {X 22.3209,Y -111.9877,Z 120,A -81.6134,B 24.9528,C -1.5874,E1 25.034,E2 527.5004} C_DIS
LIN {X 25.5998,Y -111.2821,Z 120,A -80.3677,B 24.9539,C -1.5694,E1 25.0372,E2 526.2993} C_DIS
LIN {X 28.6446,Y -110.5377,Z 120,A -78.7742,B 24.9537,C -1.5719,E1 25.0416,E2 524.7021} C_DIS
LIN {X 33.7069,Y -109.1004,Z 120,A -76.1555,B 24.9536,C -1.5739,E1 25.0486,E2 522.0832} C_DIS
LIN {X 36.6018,Y -108.1636,Z 120,A -74.6826,B 24.9536,C -1.5734,E1 25.0525,E2 520.6143} C_DIS
LIN {X 39.6442,Y -107.0873,Z 120,A -72.9322,B 24.9531,C -1.5815,E1 25.0571,E2 518.8485} C_DIS
LIN {X 43.2393,Y -105.6856,Z 120,A -70.6367,B 24.952,C -1.6006,E1 25.0632,E2 516.5129} C_DIS
LIN {X 46.57,Y -104.2613,Z 120,A -69.1903,B 24.9528,C -1.5864,E1 25.0668,E2 515.1036} C_DIS
LIN {X 49.2529,Y -103.0206,Z 120,A -67.7609,B 24.9528,C -1.5864,E1 25.0703,E2 513.6781} C_DIS
LIN {X 53.8978,Y -100.67,Z 120,A -65.0279,B 24.9523,C -1.5963,E1 25.0772,E2 510.9291} C_DIS
LIN {X 56.9185,Y -98.9915,Z 120,A -63.4724,B 24.9526,C -1.5913,E1 25.0809,E2 509.3901} C_DIS
LIN {X 59.9533,Y -97.1857,Z 120,A -61.5854,B 24.952,C -1.5999,E1 25.0854,E2 507.4887} C_DIS
LIN {X 63.1954,Y -95.1081,Z 120,A -59.7465,B 24.952,C -1.5994,E1 25.0897,E2 505.6569} C_DIS
LIN {X 66.2038,Y -93.0383,Z 120,A -57.9852,B 24.952,C -1.5999,E1 25.0937,E2 503.9005} C_DIS
LIN {X 68.7275,Y -91.19,Z 120,A -56.4062,B 24.9518,C -1.6037,E1 25.0973,E2 502.3182} C_DIS
LIN {X 70.9129,Y -89.501,Z 120,A -55.0729,B 24.9518,C -1.6043,E1 25.1002,E2 500.9884} C_DIS
LIN {X 73.2886,Y -87.567,Z 120,A -53.3737,B 24.9511,C -1.6153,E1 25.1039,E2 499.2698} C_DIS
Enddeposition()
END
